// TwinCAT 3 PLC project CorteH2y3CX9265C4
// ProgramVersion: 3.1.4024.0
// libraries:
//   CmpBitmapPool, * (System)
//   Tc2_Standard, * (Beckhoff Automation GmbH)
//   Tc2_SUPS, * (Beckhoff Automation GmbH)
//   Tc2_System, * (Beckhoff Automation GmbH)
//   Tc2_Utilities, * (Beckhoff Automation GmbH)
//   Tc3_EventLogger, * (Beckhoff Automation GmbH)
//   Tc3_Module, * (Beckhoff Automation GmbH)
//   Visu Utils, * (System)
// project tree:
//   DUTs/ StrFuncParoEnviar.TcDUT (not stored), Str_Config_ADS_to_PLC.TcDUT (not stored), Str_HistTablasMySQL.TcDUT (not stored)
//   Events_Alarms/ Eventos_PLC.TcPOU (not stored), Events.TcPOU (not stored)
//   / GlobalTextList.TcGTLO, Lectura_PLC.TcTTO, PlcTask.TcTTO, VISU_TASK.TcTTO
//   GVLs/ Fecha_PLC.TcGVL (not stored), Lectura_PLCs.TcGVL (not stored), RegistroLocalDataBase.TcGVL, Var_Com_CH2_CH3.TcGVL
//   POUs/FBs/ fbLectura_a_PLC.TcPOU (not stored), fb_Funciones_Paro.TcPOU (not stored), FuncGeneralesCortHum3.TcPOU, FuncGeneralesCortHum2.TcPOU, TempParoAcumulad.TcPOU (not stored)
//   POUs/ Fecha_Hora_PLC.TcPOU (not stored), MAIN.TcPOU
//   POUs/Funciones comunes/ Utilidades.TcPOU
//   POUs/Lectura_a_PLC_Maestro/ Lectura_Maestro.TcPOU, MAIN_Orden_Lectura_PLCs.TcPOU (not stored)
//   POUs/PRGs_Nodos/ FuncParoNodoLocalCorteH3.TcPOU, FuncParoNodoRemote1CorteH2.TcPOU
//   VISUs/ Ajustes_CorteH2.TcVIS, Ajustes_CorteH3.TcVIS, DiagnosticoFB.TcVIS, HistTablaTablas_Ch2.TcVIS, HistTablaTablas_Ch3.TcVIS, Home_CortH2.TcVIS, Home_CortH3.TcVIS, Home_Sel_Maq.TcVIS, ImagePool.TcIPO (not stored), Modelo_Tabla_Ch2.TcVIS, Modelo_Tabla_Ch3.TcVIS, VisualizationManager.TcVMO (not stored), V_Emerg_Fin_Prod_Ch2.TcVIS, V_Emerg_Fin_Prod_Ch3.TcVIS
//   VISUs/IMAGENES/ Imagenes.TcIPO (not stored)
//   VISUs/Listas_Para_Desplegables/ FormatoTabla.TcTLO, EspesorTabla.TcTLO
// real-time tasks:
//   TASK PlcTask: cycle T#10ms, priority 20, ADS port 350
//   TASK VISU_TASK: cycle T#200000us, priority 30, ADS port 351
//   TASK Lectura_PLCs: cycle T#10ms, priority 1, ADS port 352
// I/O:
//   DEVICE Device 2 (EtherCAT), AmsNetId 5.146.101.196.3.1
//     Term 1 (EK1200) [EK1200-5000 EtherCAT Power supply (2A E-Bus)]
//       Term 2 (EL1859) [EL1859 8Ch. Dig. Input 24V, 3ms, 8Ch. Dig. Output 24V, 0.5A]
//       Term 3 (EK1110) [EK1110 EtherCAT extension]
//     Term 4 (EK1100) [EK1100 EtherCAT Coupler (2A E-Bus)]
//       Term 5 (EL1859) [EL1859 8Ch. Dig. Input 24V, 3ms, 8Ch. Dig. Output 24V, 0.5A]
//       Term 6 (EL9011) [EL9011 End Terminal]
// variable links:
//   CorteH2y3CX9265C4/CorteH2y3CX9265C4 Instance <-> Device 2 (EtherCAT)/Term 1 (EK1200)/Term 2 (EL1859)
//     PlcTask Inputs/MAIN.id0Local <-> Channel 1/Input
//     PlcTask Inputs/MAIN.id0Local @bit {1..7} <-> Channel {2..8}/Input  (7 links)
//     PlcTask Outputs/MAIN.od0Local @bit {1..7} <-> Channel {10..16}/Output  (7 links)
//     PlcTask Outputs/MAIN.od0Local <-> Channel 9/Output
//   CorteH2y3CX9265C4/CorteH2y3CX9265C4 Instance <-> Device 2 (EtherCAT)/Term 4 (EK1100)/Term 5 (EL1859)
//     PlcTask Inputs/MAIN.id0Remoto1 <-> Channel 1/Input
//     PlcTask Inputs/MAIN.id0Remoto1 @bit {1..7} <-> Channel {2..8}/Input  (7 links)
//     PlcTask Outputs/MAIN.od0Remoto1 @bit {1..7} <-> Channel {10..16}/Output  (7 links)
//     PlcTask Outputs/MAIN.od0Remoto1 <-> Channel 9/Output

CONFIGURATION CorteH2y3CX9265C4
    RESOURCE PLC ON TwinCAT3
        TASK Lectura_PLC(INTERVAL := T#10ms, PRIORITY := 1);
        TASK PlcTask(INTERVAL := T#10ms, PRIORITY := 20);
        TASK VISU_TASK(INTERVAL := T#200000us, PRIORITY := 30);
        PROGRAM MAIN_Orden_Lectura_PLCs WITH Lectura_PLC : MAIN_Orden_Lectura_PLCs;
        PROGRAM MAIN WITH PlcTask : MAIN;
        PROGRAM VisuElems_Visu_Prg WITH VISU_TASK : VisuElems.Visu_Prg;
    END_RESOURCE
END_CONFIGURATION

// ---- GVLs/RegistroLocalDataBase.TcGVL
{attribute 'qualified_only'}
VAR_GLOBAL
	aValoresTurnosAnt: ARRAY [0..50] OF StrFuncParoEnviar;//Cada fin de turno se envía los valores de la ultima tabla que ha psado y se queda guardado en esta array para enseñarlo por el Scada
END_VAR
VAR_GLOBAL PERSISTENT
	//Array para el histórico de las tablas enviado a la base de datos
	 aHistoricStrTablasCH2: ARRAY[0..100]OF Str_HistTablasMySQL;
	 aHistoricStrTablasCH3: ARRAY[0..100]OF Str_HistTablasMySQL;
END_VAR

// ---- GVLs/Var_Com_CH2_CH3.TcGVL
{attribute 'qualified_only'}
VAR_GLOBAL
	// Variables Escritura en PLC Maestro 
	aStringCom AT %MW2000: ARRAY[0..97] OF STRING;	//(1 string = 81 MW)
	aWordCom AT %MW10000: ARRAY[0..249] OF WORD;	//(1 Word = 1MW)
	aBoolCom AT %MB10250: ARRAY[0..499] OF BOOL;	//(1 Bool = 1MB)
	aTimeCom AT %MW10750: ARRAY[0..124] OF TIME;	//(1 Time = 4MW)
END_VAR

// ---- POUs/MAIN.TcPOU
PROGRAM MAIN
VAR
	// UPS variables persistentes
	fbUPS: FB_S_UPS_CX81xx;//Instancia de la UPS
	// Entradas
	id0Local   AT %I*: BYTE;
	id0Remoto1 AT %I*: BYTE;
	// Salidas
	od0Local   AT %Q*: BYTE;
	od0Remoto1 AT %Q*: BYTE;
	fbUtilidades: Utilidades;
END_VAR

fbUPS(iPLCPort:= 851,);
Fecha_Hora_PLC();
Events();
fbUtilidades();
FuncParoNodoLocalCorteH3();
FuncParoNodoRemote1CorteH2();

END_PROGRAM

// ---- POUs/Funciones comunes/Utilidades.TcPOU
FUNCTION_BLOCK Utilidades
VAR_INPUT
END_VAR
VAR_OUTPUT
END_VAR
VAR
sJustificaParoComun:STRING;
END_VAR

//Direccionamiento de variables para enviar 
Var_Com_CH2_CH3.aStringCom[62] := Fecha_PLC.StringDateHourMin;

END_FUNCTION_BLOCK

// ---- POUs/PRGs_Nodos/FuncParoNodoLocalCorteH3.TcPOU
PROGRAM FuncParoNodoLocalCorteH3
VAR
	Funci_CortHum3:fb_Funciones_Paro;
	FunGeneCortHum3: FuncGeneralesCortHum3;
	//Entradas Corte húmedo 4
	Ftc_CortHum3: BOOL;	
	ForzadoFtcCortHum3:BOOL;	
	Consenso_CortHum3: BOOL;
	//Entradas fotocelula 2 libre
	Ftc2_Libre: BOOL;
	ForzadoFtc2_Libre: BOOL;
	Consenso_Ftc2_Libre: BOOL;
	//Entradas fotocelula 3 libre
	Ftc3_Libre: BOOL;
	ForzadoFtc3_Libre: BOOL;
	Consenso_Ftc3_Libre: BOOL;
	//Entradas fotocelula 4 libre
	Ftc4_Libre: BOOL;
	ForzadoFtc4_Libre: BOOL;
	Consenso_Ftc4_Libre: BOOL;
	
//	Estructuras de las variables a enviar  
	CortHum3StrFuncParoEnviar:StrFuncParoEnviar;
	Ftc2StrFuncParoEnviar:StrFuncParoEnviar;	
	Ftc3StrFuncParoEnviar:StrFuncParoEnviar;
	Ftc4StrFuncParoEnviar:StrFuncParoEnviar;
	

END_VAR
VAR_INPUT
	sFormatoEleccionTabla:STRING;
	sModeloEleccionTabla:STRING;
	sEspesorEleccionTabla:STRING;
END_VAR
VAR RETAIN
END_VAR
VAR PERSISTENT 
	HMI_Tiempo_Offset_MParo:INT:=5;
	HMI_TiempoFiltradoFotocel:TIME:=T#2S;
// Modelo de la tabla y fecha cambio de modelo
	sModeloActualTabla:STRING;
	sFormatoActualTabla:STRING;
	sEspesorActualTabla:STRING;
	sFechaInicModeloTab:STRING;


END_VAR

//Funciones de paro para cada zona(Fotocelula)

//>>>>>>>>>>>>>>>>>>>>>>>>>>>>>>>>>>>>>>>>>>>>>         	Corte húmedo 4         <<<<<<<<<<<<<<<<<<<<<<<<<<<<<<<<<<<<<<<<<<<<<<<<<<<<<<<<<<
Funci_CortHum3(Fotocelula:=Ftc_CortHum3 OR ForzadoFtcCortHum3, 
					Tiempo_Offset_MParo:=HMI_Tiempo_Offset_MParo, 
					TiempoFiltradoFotocel:=HMI_TiempoFiltradoFotocel,
					_StrFuncParoEnviar => CortHum3StrFuncParoEnviar );
					
						
						
Direccionamiento_variables_com();
LinkadoEntradas();
FunGeneCortHum3(s_ModeloActualTabla => sModeloActualTabla,
				s_ModeloEleccionTabla => sModeloEleccionTabla,
				s_FechaInicModeloTab=>sFechaInicModeloTab,
				s_FormatoActualTabla=>sFormatoActualTabla,
				s_FormatoEleccionTabla=>sFormatoEleccionTabla,
				s_EspesorActualTabla=>sEspesorActualTabla,
				s_EspesorEleccionTabla=>sEspesorEleccionTabla);

ACTION Direccionamiento_variables_com:
// Direccionamiento de las variables a la marca que les corresponde donde después se leeran desde el plc maestro



//								>>>>>>>>>>>>>>>>>>>>>>>>>>>>      WORDS    <<<<<<<<<<<<<<<<<<<<<<<<<<<<<<<<

	Var_Com_CH2_CH3.aWordCom[0]:= INT_TO_WORD (CortHum3StrFuncParoEnviar.Cont_Piezas);	    //Contadores de cada fotocelula 
	Var_Com_CH2_CH3.aWordCom[1]:= INT_TO_WORD (Ftc2StrFuncParoEnviar.Cont_Piezas);		//Contadores de cada fotocelula 
	Var_Com_CH2_CH3.aWordCom[2]:= INT_TO_WORD (Ftc3StrFuncParoEnviar.Cont_Piezas);		//Contadores de cada fotocelula 
	Var_Com_CH2_CH3.aWordCom[3]:= INT_TO_WORD (Ftc4StrFuncParoEnviar.Cont_Piezas);		//Contadores de cada fotocelula 
	Var_Com_CH2_CH3.aWordCom[4]:= INT_TO_WORD (CortHum3StrFuncParoEnviar.Min_Parado_Ftc);			//Minutos actuales parado
	Var_Com_CH2_CH3.aWordCom[5]:= INT_TO_WORD (Ftc2StrFuncParoEnviar.Min_Parado_Ftc);			//Minutos actuales parado
	Var_Com_CH2_CH3.aWordCom[6]:= INT_TO_WORD (Ftc3StrFuncParoEnviar.Min_Parado_Ftc);			//Minutos actuales parado
	Var_Com_CH2_CH3.aWordCom[7]:= INT_TO_WORD (Ftc4StrFuncParoEnviar.Min_Parado_Ftc);			//Minutos actuales parado
	
	
	
//                           	>>>>>>>>>>>>>>>>>>>>>>>>>>>>      TIME   <<<<<<<<<<<<<<<<<<<<<<<<<<<<<<<<
	
	
	Var_Com_CH2_CH3.aTimeCom[0]:=  CortHum3StrFuncParoEnviar.t_Entre_Piez_Ftc; 			//Tiempo entre piezas
	Var_Com_CH2_CH3.aTimeCom[1]:=  Ftc2StrFuncParoEnviar.t_Entre_Piez_Ftc;			//Tiempo entre piezas
	Var_Com_CH2_CH3.aTimeCom[2]:= Ftc3StrFuncParoEnviar.t_Entre_Piez_Ftc;				//Tiempo entre piezas
	Var_Com_CH2_CH3.aTimeCom[3]:= Ftc4StrFuncParoEnviar.t_Entre_Piez_Ftc;				//Tiempo entre piezas
	Var_Com_CH2_CH3.aTimeCom[4]:= CortHum3StrFuncParoEnviar.t_Entr_Piez_Ante_Ftc; 		//Tiempo entre piezas anterior
	Var_Com_CH2_CH3.aTimeCom[5]:= Ftc2StrFuncParoEnviar.t_Entr_Piez_Ante_Ftc; 		//Tiempo entre piezas anterior
	Var_Com_CH2_CH3.aTimeCom[6]:= Ftc3StrFuncParoEnviar.t_Entr_Piez_Ante_Ftc; 		//Tiempo entre piezas anterior
	Var_Com_CH2_CH3.aTimeCom[7]:= Ftc4StrFuncParoEnviar.t_Entr_Piez_Ante_Ftc; 		//Tiempo entre piezas anterior
	
	
	
	
//                           	>>>>>>>>>>>>>>>>>>>>>>>>>>>>      STRING  <<<<<<<<<<<<<<<<<<<<<<<<<<<<<<<<
    Var_Com_CH2_CH3.aStringCom[0] := CortHum3StrFuncParoEnviar.H_InParo_Ftc;         //Hora inicio paro 
	Var_Com_CH2_CH3.aStringCom[1] := Ftc2StrFuncParoEnviar.H_InParo_Ftc;         //Hora inicio paro 
	Var_Com_CH2_CH3.aStringCom[2] := Ftc3StrFuncParoEnviar.H_InParo_Ftc;         //Hora inicio paro 
	Var_Com_CH2_CH3.aStringCom[3] := Ftc4StrFuncParoEnviar.H_InParo_Ftc;         //Hora inicio paro 
	Var_Com_CH2_CH3.aStringCom[4] := CortHum3StrFuncParoEnviar.H_FinParo_Ftc;        //Hora Fin paro 
	Var_Com_CH2_CH3.aStringCom[5] := Ftc2StrFuncParoEnviar.H_FinParo_Ftc;        //Hora Fin paro 
	Var_Com_CH2_CH3.aStringCom[6] := Ftc3StrFuncParoEnviar.H_FinParo_Ftc;        //Hora Fin paro 
	Var_Com_CH2_CH3.aStringCom[7] := Ftc4StrFuncParoEnviar.H_FinParo_Ftc;        //Hora Fin paro 
	Var_Com_CH2_CH3.aStringCom[8] := CortHum3StrFuncParoEnviar.S_Justi_Paro_Ftc;		//Justificación del paro
	Var_Com_CH2_CH3.aStringCom[9] := Ftc2StrFuncParoEnviar.S_Justi_Paro_Ftc;		//Justificación del paro
	Var_Com_CH2_CH3.aStringCom[10] := Ftc3StrFuncParoEnviar.S_Justi_Paro_Ftc;		//Justificación del paro
	Var_Com_CH2_CH3.aStringCom[11] := Ftc4StrFuncParoEnviar.S_Justi_Paro_Ftc;		//Justificación del paro
	
	
//                           	>>>>>>>>>>>>>>>>>>>>>>>>>>>>      Bool  <<<<<<<<<<<<<<<<<<<<<<<<<<<<<<<<	

	Var_Com_CH2_CH3.aBoolCom[0] := CortHum3StrFuncParoEnviar.Fotocelula;						//Fotocelula Real
	Var_Com_CH2_CH3.aBoolCom[1] := Ftc2StrFuncParoEnviar.Fotocelula;						//Fotocelula Real
	Var_Com_CH2_CH3.aBoolCom[2] := Ftc3StrFuncParoEnviar.Fotocelula;						//Fotocelula Real
	Var_Com_CH2_CH3.aBoolCom[3] := Ftc4StrFuncParoEnviar.Fotocelula;						//Fotocelula Real
	Var_Com_CH2_CH3.aBoolCom[4] := CortHum3StrFuncParoEnviar.MParo_Ftc;				//Marca de paro 
	Var_Com_CH2_CH3.aBoolCom[5] := Ftc2StrFuncParoEnviar.MParo_Ftc;				//Marca de paro 
	Var_Com_CH2_CH3.aBoolCom[6] := Ftc3StrFuncParoEnviar.MParo_Ftc;				//Marca de paro 
	Var_Com_CH2_CH3.aBoolCom[7] := Ftc4StrFuncParoEnviar.MParo_Ftc;				//Marca de paro 
	Var_Com_CH2_CH3.aBoolCom[8] := CortHum3StrFuncParoEnviar.M_SinParo_Ftc;			//Marca de sin paro activo
	Var_Com_CH2_CH3.aBoolCom[9] := Ftc2StrFuncParoEnviar.M_SinParo_Ftc;			//Marca de sin paro activo
	Var_Com_CH2_CH3.aBoolCom[10] := Ftc3StrFuncParoEnviar.M_SinParo_Ftc;			//Marca de sin paro activo
	Var_Com_CH2_CH3.aBoolCom[11] := Ftc4StrFuncParoEnviar.M_SinParo_Ftc;			//Marca de sin paro activo
	Var_Com_CH2_CH3.aBoolCom[12] := CortHum3StrFuncParoEnviar.tFiltro_up_Ftc;			//Q Temp Up Filtro Fotocelulas
	Var_Com_CH2_CH3.aBoolCom[13] := Ftc2StrFuncParoEnviar.tFiltro_up_Ftc;			//Q Temp Up Filtro Fotocelulas
	Var_Com_CH2_CH3.aBoolCom[14] := Ftc3StrFuncParoEnviar.tFiltro_up_Ftc;			//Q Temp Up Filtro Fotocelulas
	Var_Com_CH2_CH3.aBoolCom[15] := Ftc4StrFuncParoEnviar.tFiltro_up_Ftc;			//Q Temp Up Filtro Fotocelulas
	Var_Com_CH2_CH3.aBoolCom[16] := CortHum3StrFuncParoEnviar.tFiltro_down_Ftc;		//Q Temp Down Filtro Fotocelulas
	Var_Com_CH2_CH3.aBoolCom[17] := Ftc2StrFuncParoEnviar.tFiltro_down_Ftc;		//Q Temp Down Filtro Fotocelulas
	Var_Com_CH2_CH3.aBoolCom[18] := Ftc3StrFuncParoEnviar.tFiltro_down_Ftc;		//Q Temp Down Filtro Fotocelulas
	Var_Com_CH2_CH3.aBoolCom[19] := Ftc4StrFuncParoEnviar.tFiltro_down_Ftc;		//Q Temp Down Filtro Fotocelulas
END_ACTION

ACTION LinkadoEntradas:
// Linkado entradas

Ftc_CortHum3:=      main.id0Local.0;
Consenso_CortHum3:= TRUE;//main.id0Remoto1.1;


Ftc2_Libre:=      main.id0Local.2;
Consenso_Ftc3_Libre:= TRUE;// main.id0Remoto1.3;


Ftc3_Libre:=      main.id0Local.4;
Consenso_Ftc3_Libre:= TRUE;// main.id0Remoto1.5;


Ftc4_Libre:=      main.id0Local.6;
Consenso_Ftc4_Libre:= TRUE;// main.id0Remoto1.7;
END_ACTION

PROPERTY PUBLIC s_JustifParoCH3 : STRING
GET
s_JustifParoCH3:= Funci_CortHum3.S_Justi_Paro_Ftc;
END_GET
SET
Funci_CortHum3.S_Justi_Paro_Ftc:=s_JustifParoCH3;
END_SET
END_PROPERTY

END_PROGRAM

// ---- POUs/FBs/FuncGeneralesCortHum3.TcPOU
FUNCTION_BLOCK FuncGeneralesCortHum3
VAR_INPUT
IndexListFormatoTabla:INT;
IndexJustificacionParo:INT;
IndexListEspesorTabla:INT;
END_VAR
VAR_OUTPUT
	//Modelo dividido en strings para DataBase
	s_ModeloActualTabla:STRING;
	s_FormatoActualTabla:STRING;
	s_EspesorActualTabla:STRING;
	s_ModeloEleccionTabla:STRING;
	s_FormatoEleccionTabla:STRING;
	s_EspesorEleccionTabla:STRING;
	//Comunes
	s_JustificaParoComun:STRING;
	s_FechaInicModeloTab:STRING;
END_VAR
VAR
	Reset_Fin_Prod:BOOL;
	P_FinProduccion:BOOL;
	P_EscribirModelo:BOOL;
	pul_Justif_Paro:BOOL;
	EscribeHistoricTablas:BOOL;
	FlancFiltUpFtcEscHistTab:R_TRIG;
	Cont1:INT;
	Cont2:INT;
	Cont3:INT;
	Cont4:INT;
END_VAR
VAR PERSISTENT 
	PointerHistTablas:INT;
END_VAR

//                             >>>>>>>>>>>>>>>> Modelo de la tabla <<<<<<<<<<<<<<<<<

//Fin de producción 		
IF P_FinProduccion THEN 
Fin_Produccion();
END_IF;
IF P_EscribirModelo THEN
	ListFormatoTabla(); 
	ListadoEspesorTabla();
	Inicio_Nuevo_Modelo();
	
END_IF


//Envío de la linea de la tabla para el historico de control producción en el HMI del operario
 IF FlancFiltUpFtcEscHistTab.Q THEN 
	 EscStrHistoricoTablas();
 END_IF


Direccionamiento_variables_com();
FlancFiltUpFtcEscHistTab(CLK := FuncParoNodoLocalCorteH3.Funci_CortHum3.tFiltro_up_Ftc.Q);

ACTION Direccionamiento_variables_com:
	//                           	>>>>>>>>>>>>>>>>>>>>>>>>>>>>      STRING      <<<<<<<<<<<<<<<<<<<<<<<<<<<<<<<<
    Var_Com_CH2_CH3.aStringCom[80] := s_ModeloActualTabla;
	Var_Com_CH2_CH3.aStringCom[81] := s_FormatoActualTabla;
	Var_Com_CH2_CH3.aStringCom[82] := s_EspesorActualTabla;
	Var_Com_CH2_CH3.aStringCom[83] := s_FechaInicModeloTab;
END_ACTION

METHOD EscStrHistoricoTablas : BOOL
VAR_INPUT
END_VAR
// Recorre todas las lineas de la tabla una posición y añade la nueva tabla en la linea 0 para mayor coodidad al visulizar

FOR PointerHistTablas := 100 TO 1 BY -1 DO 
	RegistroLocalDataBase.aHistoricStrTablasCH3[PointerHistTablas].ID := RegistroLocalDataBase.aHistoricStrTablasCH3[PointerHistTablas-1].ID;
	RegistroLocalDataBase.aHistoricStrTablasCH3[PointerHistTablas].Fecha := RegistroLocalDataBase.aHistoricStrTablasCH3[PointerHistTablas-1].Fecha;
	RegistroLocalDataBase.aHistoricStrTablasCH3[PointerHistTablas].Modelo := RegistroLocalDataBase.aHistoricStrTablasCH3[PointerHistTablas-1].Modelo;
	RegistroLocalDataBase.aHistoricStrTablasCH3[PointerHistTablas].Formato := RegistroLocalDataBase.aHistoricStrTablasCH3[PointerHistTablas-1].Formato;
	RegistroLocalDataBase.aHistoricStrTablasCH3[PointerHistTablas].Espesor :=RegistroLocalDataBase.aHistoricStrTablasCH3[PointerHistTablas-1].Espesor;
	RegistroLocalDataBase.aHistoricStrTablasCH3[PointerHistTablas].Maquina := RegistroLocalDataBase.aHistoricStrTablasCH3[PointerHistTablas-1].Maquina;
	RegistroLocalDataBase.aHistoricStrTablasCH3[PointerHistTablas].Cont_Piezas := RegistroLocalDataBase.aHistoricStrTablasCH3[PointerHistTablas-1].Cont_Piezas;
	RegistroLocalDataBase.aHistoricStrTablasCH3[PointerHistTablas].t_Entre_Piez_Ftc := RegistroLocalDataBase.aHistoricStrTablasCH3[PointerHistTablas-1].t_Entre_Piez_Ftc;
	RegistroLocalDataBase.aHistoricStrTablasCH3[PointerHistTablas].S_Justi_Paro_Ftc := RegistroLocalDataBase.aHistoricStrTablasCH3[PointerHistTablas-1].S_Justi_Paro_Ftc;
	
END_FOR
//Estructura de la array de la tabla para visualizar el historico de la tablas pasadas
RegistroLocalDataBase.aHistoricStrTablasCH3[0].ID := PointerHistTablas;
RegistroLocalDataBase.aHistoricStrTablasCH3[0].Fecha := Fecha_PLC.StringDateHourMin;
RegistroLocalDataBase.aHistoricStrTablasCH3[0].Modelo := FuncParoNodoLocalCorteH3.sModeloActualTabla;
RegistroLocalDataBase.aHistoricStrTablasCH3[0].Formato := FuncParoNodoLocalCorteH3.sFormatoActualTabla;
RegistroLocalDataBase.aHistoricStrTablasCH3[0].Espesor :=FuncParoNodoLocalCorteH3.sEspesorActualTabla;
RegistroLocalDataBase.aHistoricStrTablasCH3[0].Maquina := 'Corte húmedo 2';
RegistroLocalDataBase.aHistoricStrTablasCH3[0].Cont_Piezas := FuncParoNodoLocalCorteH3.Funci_CortHum3.Cont_Piezas_Ftc;
RegistroLocalDataBase.aHistoricStrTablasCH3[0].t_Entre_Piez_Ftc := FuncParoNodoLocalCorteH3.Funci_CortHum3.t_Entre_Piez_Ftc;
RegistroLocalDataBase.aHistoricStrTablasCH3[0].S_Justi_Paro_Ftc := FuncParoNodoLocalCorteH3.Funci_CortHum3.S_Justi_Paro_Ftc;
END_METHOD

METHOD Fin_Produccion : BOOL
VAR_INPUT	
END_VAR
var
	Puls_Fin_Produccion:BOOL;	
END_VAR
//Valores por defecto del modelo y fecha de inicio modelo

s_ModeloActualTabla:= 'Sin modelo de pieza';
s_ModeloEleccionTabla:= 'Sin modelo de pieza';
s_FormatoActualTabla:= 'Sin modelo de pieza';
s_FormatoEleccionTabla:= 'Sin modelo de pieza';
s_EspesorActualTabla:= 'Sin modelo de pieza';
s_EspesorEleccionTabla:= 'Sin modelo de pieza';
s_FechaInicModeloTab:= 'Sin modelo de pieza';
 
//Reset contador de piezas 
FuncParoNodoLocalCorteH3.Funci_CortHum3.Fin_Produccion();
END_METHOD

METHOD Inicio_Nuevo_Modelo : BOOL
VAR_INPUT
END_VAR
VAR
END_VAR

// Envías la fecha de inicio modelo de tabla 
s_FechaInicModeloTab:=Fecha_PLC.Mes_Dia_Hora_Min_Real;

//Envías el modelo de la tabla de la variable preelección  
s_ModeloActualTabla:=s_ModeloEleccionTabla;
s_FormatoActualTabla:=s_FormatoEleccionTabla;
s_EspesorActualTabla:= s_EspesorEleccionTabla;
END_METHOD

METHOD ListadoEspesorTabla : BOOL
VAR_INPUT
END_VAR
// Función para poder realizar el desplegable de espesor de la tabla en el Visu
IF IndexListEspesorTabla <> 5 THEN 
	IF IndexListEspesorTabla = 1 THEN 
		s_EspesorEleccionTabla:='3';
	END_IF
	IF IndexListEspesorTabla = 2 THEN 
		s_EspesorEleccionTabla:='6';
	END_IF
	IF IndexListEspesorTabla = 3 THEN 
		s_EspesorEleccionTabla:='12';
	END_IF
	IF IndexListEspesorTabla = 4 THEN 
		s_EspesorEleccionTabla:='20';
	END_IF
END_IF
END_METHOD

METHOD ListadoJustificacionParo : BOOL
VAR_INPUT
END_VAR
// Envío Justificación de los paros prefijados

(*Listado:  0:Sin asignar
			1: Descanso
			2: Avería
			3: Cambio de discos 
			4: Cambio de formato
			5: Cambio caballete/bandeja 
			6: Mantenimiento
			7: Falta material 
			8: Preparación material 
			9: Limpieza fin de turno 
			10: Ninguno de la lista			 
*)
//Descanso
IF IndexJustificacionParo = 1 THEN 
	FuncParoNodoLocalCorteH3.s_JustifParoCH3 := 'Descanso';
END_IF
// Avería 
IF IndexJustificacionParo = 2 THEN 
	FuncParoNodoLocalCorteH3.s_JustifParoCH3 := 'Avería';
END_IF
//Cambio de discos 
IF IndexJustificacionParo = 3 THEN 
	FuncParoNodoLocalCorteH3.s_JustifParoCH3 := 'Cambio de discos';
END_IF
// Cambio de formato
IF IndexJustificacionParo = 4 THEN 
	FuncParoNodoLocalCorteH3.s_JustifParoCH3 := 'Cambio de formato';
END_IF
//Cambio caballete/bandeja
IF IndexJustificacionParo = 5 THEN 
	FuncParoNodoLocalCorteH3.s_JustifParoCH3 := 'Cambio caballete/bandeja';
END_IF
// Mantenimiento
IF IndexJustificacionParo = 6 THEN 
	FuncParoNodoLocalCorteH3.s_JustifParoCH3 := 'Mantenimiento';
END_IF
// Falta de material 
IF IndexJustificacionParo = 7 THEN 
	FuncParoNodoLocalCorteH3.s_JustifParoCH3 := 'Falta de material';
END_IF
//Preparación de material 
IF IndexJustificacionParo = 8 THEN 
	FuncParoNodoLocalCorteH3.s_JustifParoCH3 := 'Preparación de material';
END_IF
// Limpieza fin de turno
IF IndexJustificacionParo = 9 THEN 
	FuncParoNodoLocalCorteH3.s_JustifParoCH3 := 'Limpieza fin de turno';
END_IF
// No está en la lista
IF IndexJustificacionParo = 10 THEN 
	FuncParoNodoLocalCorteH3.s_JustifParoCH3 := 'ESCRIBE AQUÍ LA JUSTIFICACIÓN DEL PARO';
END_IF
END_METHOD

METHOD ListFormatoTabla : BOOL
VAR_INPUT
END_VAR
// Función para poder realizar el desplegable de formato de la tabla en el Visu
IF IndexListFormatoTabla <> 8 THEN 
	IF IndexListFormatoTabla = 1 THEN 
		s_FormatoEleccionTabla:='3200 X 1500';
		Cont1:=Cont1+1;
	END_IF
	IF IndexListFormatoTabla = 2 THEN 
		s_FormatoEleccionTabla:='3600 X 1200';
		Cont2:=Cont2+1;
	END_IF
	IF IndexListFormatoTabla = 3 THEN 
		s_FormatoEleccionTabla:='1800 X 1200';
	END_IF
	IF IndexListFormatoTabla = 4 THEN 
		s_FormatoEleccionTabla:='3000 X 1000';
	END_IF
	IF IndexListFormatoTabla = 5 THEN 
		s_FormatoEleccionTabla:='2600 X 1500';
	END_IF
	IF IndexListFormatoTabla = 6 THEN 
		s_FormatoEleccionTabla:='800 X 700';
	END_IF
	IF IndexListFormatoTabla = 7 THEN 
		s_FormatoEleccionTabla:='2700 X 1000';
	END_IF
END_IF
END_METHOD

END_FUNCTION_BLOCK

// ---- POUs/PRGs_Nodos/FuncParoNodoRemote1CorteH2.TcPOU
PROGRAM FuncParoNodoRemote1CorteH2
VAR
	Funci_CortHum2:fb_Funciones_Paro;
	FunGeneCortHum2: FuncGeneralesCortHum2;
	//Entradas Corte húmedo 4
	Ftc_CortHum2: BOOL;	
	ForzadoFtcCortHum2:BOOL;	
	Consenso_CortHum2: BOOL;
	//Entradas fotocelula 2 libre
	Ftc2_Libre: BOOL;
	ForzadoFtc2_Libre: BOOL;
	Consenso_Ftc2_Libre: BOOL;
	//Entradas fotocelula 3 libre
	Ftc3_Libre: BOOL;
	ForzadoFtc3_Libre: BOOL;
	Consenso_Ftc3_Libre: BOOL;
	//Entradas fotocelula 4 libre
	Ftc4_Libre: BOOL;
	ForzadoFtc4_Libre: BOOL;
	Consenso_Ftc4_Libre: BOOL;
	
//	Estructuras de las variables a enviar  
	CortHum2StrFuncParoEnviar:StrFuncParoEnviar;
	Ftc2StrFuncParoEnviar:StrFuncParoEnviar;	
	Ftc3StrFuncParoEnviar:StrFuncParoEnviar;
	Ftc4StrFuncParoEnviar:StrFuncParoEnviar;
	

END_VAR
VAR_INPUT
	sFormatoEleccionTabla:STRING;
	sModeloEleccionTabla:STRING;
	sEspesorEleccionTabla:STRING;
END_VAR
VAR RETAIN
END_VAR
VAR PERSISTENT 
	HMI_Tiempo_Offset_MParo:INT:=5;
	HMI_TiempoFiltradoFotocel:TIME:=T#2S;
// Modelo de la tabla y fecha cambio de modelo
	sModeloActualTabla:STRING;
	sFormatoActualTabla:STRING;
	sEspesorActualTabla:STRING;
	sFechaInicModeloTab:STRING;


END_VAR

//Funciones de paro para cada zona(Fotocelula)

//>>>>>>>>>>>>>>>>>>>>>>>>>>>>>>>>>>>>>>>>>>>>>         	Corte húmedo 4         <<<<<<<<<<<<<<<<<<<<<<<<<<<<<<<<<<<<<<<<<<<<<<<<<<<<<<<<<<
Funci_CortHum2(Fotocelula:=Ftc_CortHum2 OR ForzadoFtcCortHum2, 
					Tiempo_Offset_MParo:=HMI_Tiempo_Offset_MParo, 
					TiempoFiltradoFotocel:=HMI_TiempoFiltradoFotocel,
					_StrFuncParoEnviar => CortHum2StrFuncParoEnviar );
					
						
						
Direccionamiento_variables_com();
LinkadoEntradas();
FunGeneCortHum2(s_ModeloActualTabla => sModeloActualTabla,s_ModeloEleccionTabla => sModeloEleccionTabla,s_FechaInicModeloTab=>sFechaInicModeloTab,s_FormatoActualTabla=>sFormatoActualTabla,s_FormatoEleccionTabla=>sFormatoEleccionTabla,s_EspesorActualTabla=>sEspesorActualTabla,s_EspesorEleccionTabla=>sEspesorEleccionTabla);

ACTION Direccionamiento_variables_com:
// Direccionamiento de las variables a la marca que les corresponde donde despés se leeran desde el plc maestro



//								>>>>>>>>>>>>>>>>>>>>>>>>>>>>      WORDS    <<<<<<<<<<<<<<<<<<<<<<<<<<<<<<<<

	Var_Com_CH2_CH3.aWordCom[50]:= INT_TO_WORD (CortHum2StrFuncParoEnviar.Cont_Piezas);	    //Contadores de cada fotocelula 
	Var_Com_CH2_CH3.aWordCom[51]:= INT_TO_WORD (Ftc2StrFuncParoEnviar.Cont_Piezas);		//Contadores de cada fotocelula 
	Var_Com_CH2_CH3.aWordCom[52]:= INT_TO_WORD (Ftc3StrFuncParoEnviar.Cont_Piezas);		//Contadores de cada fotocelula 
	Var_Com_CH2_CH3.aWordCom[53]:= INT_TO_WORD (Ftc4StrFuncParoEnviar.Cont_Piezas);		//Contadores de cada fotocelula 
	Var_Com_CH2_CH3.aWordCom[54]:= INT_TO_WORD (CortHum2StrFuncParoEnviar.Min_Parado_Ftc);			//Minutos actuales parado
	Var_Com_CH2_CH3.aWordCom[55]:= INT_TO_WORD (Ftc2StrFuncParoEnviar.Min_Parado_Ftc);			//Minutos actuales parado
	Var_Com_CH2_CH3.aWordCom[56]:= INT_TO_WORD (Ftc3StrFuncParoEnviar.Min_Parado_Ftc);			//Minutos actuales parado
	Var_Com_CH2_CH3.aWordCom[57]:= INT_TO_WORD (Ftc4StrFuncParoEnviar.Min_Parado_Ftc);			//Minutos actuales parado
	
	
	
//                           	>>>>>>>>>>>>>>>>>>>>>>>>>>>>      TIME   <<<<<<<<<<<<<<<<<<<<<<<<<<<<<<<<
	
	
	Var_Com_CH2_CH3.aTimeCom[25]:=  CortHum2StrFuncParoEnviar.t_Entre_Piez_Ftc; 			//Tiempo entre piezas
	Var_Com_CH2_CH3.aTimeCom[26]:=  Ftc2StrFuncParoEnviar.t_Entre_Piez_Ftc;			//Tiempo entre piezas
	Var_Com_CH2_CH3.aTimeCom[27]:= Ftc3StrFuncParoEnviar.t_Entre_Piez_Ftc;				//Tiempo entre piezas
	Var_Com_CH2_CH3.aTimeCom[28]:= Ftc4StrFuncParoEnviar.t_Entre_Piez_Ftc;				//Tiempo entre piezas
	Var_Com_CH2_CH3.aTimeCom[29]:= CortHum2StrFuncParoEnviar.t_Entr_Piez_Ante_Ftc; 		//Tiempo entre piezas anterior
	Var_Com_CH2_CH3.aTimeCom[30]:= Ftc2StrFuncParoEnviar.t_Entr_Piez_Ante_Ftc; 		//Tiempo entre piezas anterior
	Var_Com_CH2_CH3.aTimeCom[31]:= Ftc3StrFuncParoEnviar.t_Entr_Piez_Ante_Ftc; 		//Tiempo entre piezas anterior
	Var_Com_CH2_CH3.aTimeCom[32]:= Ftc4StrFuncParoEnviar.t_Entr_Piez_Ante_Ftc; 		//Tiempo entre piezas anterior
	
	
	
	
//                           	>>>>>>>>>>>>>>>>>>>>>>>>>>>>      STRING  <<<<<<<<<<<<<<<<<<<<<<<<<<<<<<<<
    Var_Com_CH2_CH3.aStringCom[20] := CortHum2StrFuncParoEnviar.H_InParo_Ftc;         //Hora inicio paro 
	Var_Com_CH2_CH3.aStringCom[21] := Ftc2StrFuncParoEnviar.H_InParo_Ftc;         //Hora inicio paro 
	Var_Com_CH2_CH3.aStringCom[22] := Ftc3StrFuncParoEnviar.H_InParo_Ftc;         //Hora inicio paro 
	Var_Com_CH2_CH3.aStringCom[23] := Ftc4StrFuncParoEnviar.H_InParo_Ftc;         //Hora inicio paro 
	Var_Com_CH2_CH3.aStringCom[24] := CortHum2StrFuncParoEnviar.H_FinParo_Ftc;        //Hora Fin paro 
	Var_Com_CH2_CH3.aStringCom[25] := Ftc2StrFuncParoEnviar.H_FinParo_Ftc;        //Hora Fin paro 
	Var_Com_CH2_CH3.aStringCom[26] := Ftc3StrFuncParoEnviar.H_FinParo_Ftc;        //Hora Fin paro 
	Var_Com_CH2_CH3.aStringCom[27] := Ftc4StrFuncParoEnviar.H_FinParo_Ftc;        //Hora Fin paro 
	Var_Com_CH2_CH3.aStringCom[28] := CortHum2StrFuncParoEnviar.S_Justi_Paro_Ftc;		//Justificación del paro
	Var_Com_CH2_CH3.aStringCom[29] := Ftc2StrFuncParoEnviar.S_Justi_Paro_Ftc;		//Justificación del paro
	Var_Com_CH2_CH3.aStringCom[30] := Ftc3StrFuncParoEnviar.S_Justi_Paro_Ftc;		//Justificación del paro
	Var_Com_CH2_CH3.aStringCom[31] := Ftc4StrFuncParoEnviar.S_Justi_Paro_Ftc;		//Justificación del paro
	
	
//                           	>>>>>>>>>>>>>>>>>>>>>>>>>>>>      Bool  <<<<<<<<<<<<<<<<<<<<<<<<<<<<<<<<	

	Var_Com_CH2_CH3.aBoolCom[99] := CortHum2StrFuncParoEnviar.Fotocelula;						//Fotocelula Real
	Var_Com_CH2_CH3.aBoolCom[100] := Ftc2StrFuncParoEnviar.Fotocelula;						//Fotocelula Real
	Var_Com_CH2_CH3.aBoolCom[101] := Ftc3StrFuncParoEnviar.Fotocelula;						//Fotocelula Real
	Var_Com_CH2_CH3.aBoolCom[102] := Ftc4StrFuncParoEnviar.Fotocelula;						//Fotocelula Real
	Var_Com_CH2_CH3.aBoolCom[103] := CortHum2StrFuncParoEnviar.MParo_Ftc;				//Marca de paro 
	Var_Com_CH2_CH3.aBoolCom[104] := Ftc2StrFuncParoEnviar.MParo_Ftc;				//Marca de paro 
	Var_Com_CH2_CH3.aBoolCom[105] := Ftc3StrFuncParoEnviar.MParo_Ftc;				//Marca de paro 
	Var_Com_CH2_CH3.aBoolCom[106] := Ftc4StrFuncParoEnviar.MParo_Ftc;				//Marca de paro 
	Var_Com_CH2_CH3.aBoolCom[107] := CortHum2StrFuncParoEnviar.M_SinParo_Ftc;			//Marca de sin paro activo
	Var_Com_CH2_CH3.aBoolCom[108] := Ftc2StrFuncParoEnviar.M_SinParo_Ftc;			//Marca de sin paro activo
	Var_Com_CH2_CH3.aBoolCom[109] := Ftc3StrFuncParoEnviar.M_SinParo_Ftc;			//Marca de sin paro activo
	Var_Com_CH2_CH3.aBoolCom[110] := Ftc4StrFuncParoEnviar.M_SinParo_Ftc;			//Marca de sin paro activo
	Var_Com_CH2_CH3.aBoolCom[111] := CortHum2StrFuncParoEnviar.tFiltro_up_Ftc;			//Q Temp Up Filtro Fotocelulas
	Var_Com_CH2_CH3.aBoolCom[112] := Ftc2StrFuncParoEnviar.tFiltro_up_Ftc;			//Q Temp Up Filtro Fotocelulas
	Var_Com_CH2_CH3.aBoolCom[113] := Ftc3StrFuncParoEnviar.tFiltro_up_Ftc;			//Q Temp Up Filtro Fotocelulas
	Var_Com_CH2_CH3.aBoolCom[114] := Ftc4StrFuncParoEnviar.tFiltro_up_Ftc;			//Q Temp Up Filtro Fotocelulas
	Var_Com_CH2_CH3.aBoolCom[115] := CortHum2StrFuncParoEnviar.tFiltro_down_Ftc;		//Q Temp Down Filtro Fotocelulas
	Var_Com_CH2_CH3.aBoolCom[116] := Ftc2StrFuncParoEnviar.tFiltro_down_Ftc;		//Q Temp Down Filtro Fotocelulas
	Var_Com_CH2_CH3.aBoolCom[117] := Ftc3StrFuncParoEnviar.tFiltro_down_Ftc;		//Q Temp Down Filtro Fotocelulas
	Var_Com_CH2_CH3.aBoolCom[118] := Ftc4StrFuncParoEnviar.tFiltro_down_Ftc;		//Q Temp Down Filtro Fotocelulas
END_ACTION

ACTION LinkadoEntradas:





// Linkado entradas

Ftc_CortHum2:=      main.id0Remoto1.0;
Consenso_CortHum2:= TRUE;//main.id0Remoto1.1;


Ftc2_Libre:=      main.id0Remoto1.2;
Consenso_Ftc3_Libre:= TRUE;// main.id0Remoto1.3;


Ftc3_Libre:=      main.id0Remoto1.4;
Consenso_Ftc3_Libre:= TRUE;// main.id0Remoto1.5;


Ftc4_Libre:=      main.id0Remoto1.6;
Consenso_Ftc4_Libre:= TRUE;// main.id0Remoto1.7;
END_ACTION

PROPERTY PUBLIC s_JustifParoCH2 : STRING
GET
s_JustifParoCH2:= Funci_CortHum2.S_Justi_Paro_Ftc;
END_GET
SET
Funci_CortHum2.S_Justi_Paro_Ftc:=s_JustifParoCH2;
END_SET
END_PROPERTY

END_PROGRAM

// ---- POUs/FBs/FuncGeneralesCortHum2.TcPOU
FUNCTION_BLOCK FuncGeneralesCortHum2
VAR_INPUT
IndexListFormatoTabla:INT;
IndexJustificacionParo:INT;
IndexListEspesorTabla:INT;
END_VAR
VAR_OUTPUT
	//Modelo dividido en strings para DataBase
	s_ModeloActualTabla:STRING;
	s_FormatoActualTabla:STRING;
	s_EspesorActualTabla:STRING;
	s_ModeloEleccionTabla:STRING;
	s_FormatoEleccionTabla:STRING;
	s_EspesorEleccionTabla:STRING;
	//Comunes
	s_JustificaParoComun:STRING;
	s_FechaInicModeloTab:STRING;
END_VAR
VAR
	Reset_Fin_Prod:BOOL;
	P_FinProduccion:BOOL;
	P_EscribirModelo:BOOL;
	pul_Justif_Paro:BOOL;
	EscribeHistoricTablas:BOOL;
	FlancFiltUpFtcEscHistTab:R_TRIG;
	Cont1:INT;
	Cont2:INT;
	Cont3:INT;
	Cont4:INT;
END_VAR
VAR PERSISTENT 
	PointerHistTablas:INT;
END_VAR

//                             >>>>>>>>>>>>>>>> Modelo de la tabla <<<<<<<<<<<<<<<<<

//Fin de producción 		
IF P_FinProduccion THEN 
Fin_Produccion();
END_IF;
IF P_EscribirModelo THEN
	ListFormatoTabla(); 
	ListadoEspesorTabla();
	Inicio_Nuevo_Modelo();
	
END_IF


//Envío de la linea de la tabla para el historico de control producción en el HMI del operario
 IF FlancFiltUpFtcEscHistTab.Q THEN 
	 EscStrHistoricoTablas();
 END_IF


Direccionamiento_variables_com();
FlancFiltUpFtcEscHistTab(CLK := FuncParoNodoRemote1CorteH2.Funci_CortHum2.tFiltro_up_Ftc.Q);

ACTION Direccionamiento_variables_com:
	//                           	>>>>>>>>>>>>>>>>>>>>>>>>>>>>      STRING      <<<<<<<<<<<<<<<<<<<<<<<<<<<<<<<<
    Var_Com_CH2_CH3.aStringCom[84] := s_ModeloActualTabla;
	Var_Com_CH2_CH3.aStringCom[85] := s_FormatoActualTabla;
	Var_Com_CH2_CH3.aStringCom[86] := s_EspesorActualTabla;
	Var_Com_CH2_CH3.aStringCom[87] := s_FechaInicModeloTab;
END_ACTION

METHOD EscStrHistoricoTablas : BOOL
VAR_INPUT
END_VAR
// Recorre todas las lineas de la tabla una posición y añade la nueva tabla en la linea 0 para mayor coodidad al visulizar

FOR PointerHistTablas := 100 TO 1 BY -1 DO 
	RegistroLocalDataBase.aHistoricStrTablasCH2[PointerHistTablas].ID := RegistroLocalDataBase.aHistoricStrTablasCH2[PointerHistTablas-1].ID;
	RegistroLocalDataBase.aHistoricStrTablasCH2[PointerHistTablas].Fecha := RegistroLocalDataBase.aHistoricStrTablasCH2[PointerHistTablas-1].Fecha;
	RegistroLocalDataBase.aHistoricStrTablasCH2[PointerHistTablas].Modelo := RegistroLocalDataBase.aHistoricStrTablasCH2[PointerHistTablas-1].Modelo;
	RegistroLocalDataBase.aHistoricStrTablasCH2[PointerHistTablas].Formato := RegistroLocalDataBase.aHistoricStrTablasCH2[PointerHistTablas-1].Formato;
	RegistroLocalDataBase.aHistoricStrTablasCH2[PointerHistTablas].Espesor :=RegistroLocalDataBase.aHistoricStrTablasCH2[PointerHistTablas-1].Espesor;
	RegistroLocalDataBase.aHistoricStrTablasCH2[PointerHistTablas].Maquina := RegistroLocalDataBase.aHistoricStrTablasCH2[PointerHistTablas-1].Maquina;
	RegistroLocalDataBase.aHistoricStrTablasCH2[PointerHistTablas].Cont_Piezas := RegistroLocalDataBase.aHistoricStrTablasCH2[PointerHistTablas-1].Cont_Piezas;
	RegistroLocalDataBase.aHistoricStrTablasCH2[PointerHistTablas].t_Entre_Piez_Ftc := RegistroLocalDataBase.aHistoricStrTablasCH2[PointerHistTablas-1].t_Entre_Piez_Ftc;
	RegistroLocalDataBase.aHistoricStrTablasCH2[PointerHistTablas].S_Justi_Paro_Ftc := RegistroLocalDataBase.aHistoricStrTablasCH2[PointerHistTablas-1].S_Justi_Paro_Ftc;
	
END_FOR
//Estructura de la array de la tabla para visualizar el historico de la tablas pasadas
RegistroLocalDataBase.aHistoricStrTablasCH2[0].ID := PointerHistTablas;
RegistroLocalDataBase.aHistoricStrTablasCH2[0].Fecha := Fecha_PLC.StringDateHourMin;
RegistroLocalDataBase.aHistoricStrTablasCH2[0].Modelo := FuncParoNodoRemote1CorteH2.sModeloActualTabla;
RegistroLocalDataBase.aHistoricStrTablasCH2[0].Formato := FuncParoNodoRemote1CorteH2.sFormatoActualTabla;
RegistroLocalDataBase.aHistoricStrTablasCH2[0].Espesor :=FuncParoNodoRemote1CorteH2.sEspesorActualTabla;
RegistroLocalDataBase.aHistoricStrTablasCH2[0].Maquina := 'Corte húmedo 2';
RegistroLocalDataBase.aHistoricStrTablasCH2[0].Cont_Piezas := FuncParoNodoRemote1CorteH2.Funci_CortHum2.Cont_Piezas_Ftc;
RegistroLocalDataBase.aHistoricStrTablasCH2[0].t_Entre_Piez_Ftc := FuncParoNodoRemote1CorteH2.Funci_CortHum2.t_Entre_Piez_Ftc;
RegistroLocalDataBase.aHistoricStrTablasCH2[0].S_Justi_Paro_Ftc := FuncParoNodoRemote1CorteH2.Funci_CortHum2.S_Justi_Paro_Ftc;
END_METHOD

METHOD Fin_Produccion : BOOL
VAR_INPUT	
END_VAR
var
	Puls_Fin_Produccion:BOOL;	
END_VAR
//Valores por defecto del modelo y fecha de inicio modelo

s_ModeloActualTabla:= 'Sin modelo de pieza';
s_ModeloEleccionTabla:= 'Sin modelo de pieza';
s_FormatoActualTabla:= 'Sin modelo de pieza';
s_FormatoEleccionTabla:= 'Sin modelo de pieza';
s_EspesorActualTabla:= 'Sin modelo de pieza';
s_EspesorEleccionTabla:= 'Sin modelo de pieza';
s_FechaInicModeloTab:= 'Sin modelo de pieza';
 
//Reset contador de piezas 
FuncParoNodoRemote1CorteH2.Funci_CortHum2.Fin_Produccion();
END_METHOD

METHOD Inicio_Nuevo_Modelo : BOOL
VAR_INPUT
END_VAR
VAR
END_VAR

// Envías la fecha de inicio modelo de tabla 
s_FechaInicModeloTab:=Fecha_PLC.Mes_Dia_Hora_Min_Real;

//Envías el modelo de la tabla de la variable preelección  
s_ModeloActualTabla:=s_ModeloEleccionTabla;
s_FormatoActualTabla:=s_FormatoEleccionTabla;
s_EspesorActualTabla:= s_EspesorEleccionTabla;
END_METHOD

METHOD ListadoEspesorTabla : BOOL
VAR_INPUT
END_VAR
// Función para poder realizar el desplegable de espesor de la tabla en el Visu
IF IndexListEspesorTabla <> 5 THEN 
	IF IndexListEspesorTabla = 1 THEN 
		s_EspesorEleccionTabla:='3';
	END_IF
	IF IndexListEspesorTabla = 2 THEN 
		s_EspesorEleccionTabla:='6';
	END_IF
	IF IndexListEspesorTabla = 3 THEN 
		s_EspesorEleccionTabla:='12';
	END_IF
	IF IndexListEspesorTabla = 4 THEN 
		s_EspesorEleccionTabla:='20';
	END_IF
END_IF
END_METHOD

METHOD ListadoJustificacionParo : BOOL
VAR_INPUT
END_VAR
// Envío Justificación de los paros prefijados

(*Listado:  0:Sin asignar
			1: Descanso
			2: Avería
			3: Cambio de discos 
			4: Cambio de formato
			5: Cambio caballete/bandeja 
			6: Mantenimiento
			7: Falta material 
			8: Preparación material 
			9: Limpieza fin de turno 
			10: Ninguno de la lista			 
*)
//Descanso
IF IndexJustificacionParo = 1 THEN 
	FuncParoNodoRemote1CorteH2.s_JustifParoCH2 := 'Descanso';
END_IF
// Avería 
IF IndexJustificacionParo = 2 THEN 
	FuncParoNodoRemote1CorteH2.s_JustifParoCH2 := 'Avería';
END_IF
//Cambio de discos 
IF IndexJustificacionParo = 3 THEN 
	FuncParoNodoRemote1CorteH2.s_JustifParoCH2 := 'Cambio de discos';
END_IF
// Cambio de formato
IF IndexJustificacionParo = 4 THEN 
	FuncParoNodoRemote1CorteH2.s_JustifParoCH2 := 'Cambio de formato';
END_IF
//Cambio caballete/bandeja
IF IndexJustificacionParo = 5 THEN 
	FuncParoNodoRemote1CorteH2.s_JustifParoCH2 := 'Cambio caballete/bandeja';
END_IF
// Mantenimiento
IF IndexJustificacionParo = 6 THEN 
	FuncParoNodoRemote1CorteH2.s_JustifParoCH2 := 'Mantenimiento';
END_IF
// Falta de material 
IF IndexJustificacionParo = 7 THEN 
	FuncParoNodoRemote1CorteH2.s_JustifParoCH2 := 'Falta de material';
END_IF
//Preparación de material 
IF IndexJustificacionParo = 8 THEN 
	FuncParoNodoRemote1CorteH2.s_JustifParoCH2 := 'Preparación de material';
END_IF
// Limpieza fin de turno
IF IndexJustificacionParo = 9 THEN 
	FuncParoNodoRemote1CorteH2.s_JustifParoCH2 := 'Limpieza fin de turno';
END_IF
// No está en la lista
IF IndexJustificacionParo = 10 THEN 
	FuncParoNodoRemote1CorteH2.s_JustifParoCH2 := 'ESCRIBE AQUÍ LA JUSTIFICACIÓN DEL PARO';
END_IF
END_METHOD

METHOD ListFormatoTabla : BOOL
VAR_INPUT
END_VAR
// Función para poder realizar el desplegable de formato de la tabla en el Visu
IF IndexListFormatoTabla <> 8 THEN 
	IF IndexListFormatoTabla = 1 THEN 
		s_FormatoEleccionTabla:='3200 X 1500';
		Cont1:=Cont1+1;
	END_IF
	IF IndexListFormatoTabla = 2 THEN 
		s_FormatoEleccionTabla:='3600 X 1200';
		Cont2:=Cont2+1;
	END_IF
	IF IndexListFormatoTabla = 3 THEN 
		s_FormatoEleccionTabla:='1800 X 1200';
	END_IF
	IF IndexListFormatoTabla = 4 THEN 
		s_FormatoEleccionTabla:='3000 X 1000';
	END_IF
	IF IndexListFormatoTabla = 5 THEN 
		s_FormatoEleccionTabla:='2600 X 1500';
	END_IF
	IF IndexListFormatoTabla = 6 THEN 
		s_FormatoEleccionTabla:='800 X 700';
	END_IF
	IF IndexListFormatoTabla = 7 THEN 
		s_FormatoEleccionTabla:='2700 X 1000';
	END_IF
END_IF
END_METHOD

END_FUNCTION_BLOCK

// ---- POUs/Lectura_a_PLC_Maestro/Lectura_Maestro.TcPOU
PROGRAM Lectura_Maestro
VAR
	// >>>>>>>>>>>>>>>>>>>>>>>>>>>>>>>>>>>>>>>>   Estructuras de configuración con la comunicación desde y hacia el PLC Maestro <<<<<<<<<<<<<<<<<<<<<<<<<<<<<<<<<<<<<<<<<<<<<<<<<
	
	//Recordar que el IDXOFFS debe ser el doble de la posición a la que queréis acceder Ejemplo: para leer los strings a partir de la dirección MW100 Debéis poner 200 en exadecimal (C8)
	
//Configuración de la lectura de las variables Bool, IDXGRP:=16#4020(Hace referencia a la lectura de M),IDXOFFS:=16#B48C(Offset %MB46.220,  %MB46.220 a %MB46320), LEN : 101 Longitud bools leidos,DESTADDR:= ADR(Lectura_PLCs.aMasterBoolCom) Ubicación del array donde se guarda la lectura
	Config_Read_ADS_Bools_Maestro:Str_Config_ADS_to_PLC:=(NETID:='192.168.10.71.1.1', PORT:=851, IDXGRP:=16#4020,IDXOFFS:=16#B48C,LEN:=101,DESTADDR:= ADR(Lectura_PLCs.aMasterBoolCom));
	
	//Configuración de la lectura de las variables String, IDXGRP:=16#4020(Hace referencia a la lectura de M),IDXOFFS:= 16#14500(%MW42600 a %MW43815 ( 15 word)),Longitud de bytes a leer 1215 bytes = 15 strings que son 81words por cada string. ,DESTADDR:= ADR(Lectura_PLCs.aMasterStringCom) Ubicación del array donde se guarda la lectura
	Config_Read_ADS_Strings_Maestro:Str_Config_ADS_to_PLC:=(NETID:='192.168.10.71.1.1', PORT:=851, IDXGRP:=16#4020,IDXOFFS:=16#14500,LEN:=1215,DESTADDR:= ADR(Lectura_PLCs.aMasterStringCom));
	
	//Configuración de la lectura de las variables Times, IDXGRP:=16#4020(Hace referencia a la lectura de M),IDXOFFS:=16#17278 ( %MW47420 a %MW47614 (204 word),LEN:= 204 Longitud de bytes a leer bytes = 200words    51 componentes,DESTADDR:= ADR(Lectura_PLCs.aMasterTimeCom) Ubicación del array donde se guarda la lectura
	Config_Read_ADS_Times_Maestro:Str_Config_ADS_to_PLC:=(NETID:='192.168.10.71.1.1', PORT:=851, IDXGRP:=16#4020,IDXOFFS:=16#17278,LEN:= 204,DESTADDR:= ADR(Lectura_PLCs.aMasterTimeCom));
	
	//Configuración de la lectura de las variables Words, IDXGRP:=16#4020(Hace referencia a la lectura de M),IDXOFFS:=16#16008 ( %MW45060 a %MW45100 (40 word),82;//Longitud de bytes a leer 80 bytes = 40words   ,DESTADDR:= ADR(Lectura_PLCs.aMasteWordCom) Ubicación del array donde se guarda la lectura
	Config_Read_ADS_Words_Maestro:Str_Config_ADS_to_PLC:=(NETID:='192.168.10.71.1.1', PORT:=851, IDXGRP:=16#4020,IDXOFFS:=16#16008,LEN:=82,DESTADDR:= ADR(Lectura_PLCs.aMasterWordCom));
	
	fbLectura_a_PLC_Maestro:fbLectura_a_PLC;
	

END_VAR
VAR_INPUT
	bNextBlockToRead_L4_Done:BOOL;
END_VAR

fbLectura_a_PLC_Maestro(
	Config_PLC_ADS_Bools:=Config_Read_ADS_Bools_Maestro,
	Config_PLC_ADS_Strings:=Config_Read_ADS_Strings_Maestro,
	Config_PLC_ADS_Times:=Config_Read_ADS_Times_Maestro,
	Config_PLC_ADS_Words:=Config_Read_ADS_Words_Maestro,
 	TimeReadStateEntreLecturas:=T#20MS,
	bHabilitadaLectura:=TRUE,
	);

END_PROGRAM

// ---- GlobalTextList.TcGTLO
TEXTLIST GlobalTextList
  505 = '%i'
  650 = '%s'
  177 = '%s \tContador piezas corte húmedo 4 '
  771 = '%s \tContador piezas Multidiscos 2'
  56 = "%t[H'h'm'min']"
  702 = '%t[HH,mm]'
  1013 = '%t[HH:mm]h'
  410 = '%t[HHmm]'
  696 = '%t[H]h[m]min'
  175 = '%t[min]'
  633 = '%t[s,ms]'
  1163 = 'ACEPTAR'
  1790 = 'AJUSTE\nMEDIDAS/PRECORTE'
  152 = 'Ajustes'
  636 = 'Atrás'
  589 = 'AVERÍA'
  1710 = 'CAMBIO \nCABALLETE/BANDEJA'
  1137 = 'CAMBIO DISCOS'
  288 = 'CAMBIO FORMATO'
  856 = 'Contador de piezas'
  115 = 'Corte húmedo 2'
  548 = 'CORTE HÚMEDO 2'
  979 = 'Corte húmedo 3'
  913 = 'CORTE HÚMEDO 3'
  137 = 'Corte húmedo 4'
  1186 = 'CORTE HÚMEDO 4'
  952 = 'Decoración'
  448 = 'Delay Escritura'
  1310 = 'DESCANSO'
  503 = 'Diagnóstico lineas'
  1366 = 'Día'
  765 = 'Elige la línea la cual quieres ver el estado de sus contadores y señales'
  630 = 'En producción'
  432 = 'En producción todo OK'
  331 = 'En produccoón desde:    %s'
  434 = 'Entrada Horno Inferior '
  370 = 'Entrada Horno Superior'
  557 = 'Entrada secadero'
  466 = 'Entre Piez %s'
  850 = 'Entre Piez Anterior %s'
  740 = 'ESPESOR'
  631 = 'Espesor'
  818 = 'Exit'
  1436 = 'FALTA DE MATERIAL'
  1029 = 'Fecha'
  394 = 'Fecha inicio del modelo actual'
  297 = 'Filtro Down'
  866 = 'Filtro Up'
  796 = 'Fin de producción del modelo'
  766 = 'FINALIZAR MODELO'
  79 = 'FORMATO'
  419 = 'Formato'
  884 = 'Forzar Fotocelula'
  768 = 'Habilitar escritura \nen MySQL'
  350 = 'Habilitar escritura Linea 4\nen MySQL'
  841 = 'Habilitar lectura a\nPLC L4'
  332 = 'Habilitar lectura a\nPLCs'
  34 = 'Habilitar lectura al\nPLC Maestro'
  907 = 'HISTÓRICO'
  532 = 'Histórico'
  248 = 'HISTÓRICO PRODUCCIÓN'
  689 = 'Home'
  681 = 'Hora Fin Paro'
  1204 = 'HORA INICIO'
  553 = 'Hora Inicio del paro'
  340 = 'Hora Inicio Paro'
  358 = 'Horno Inf.'
  962 = 'Horno Sup.'
  733 = 'ID'
  867 = 'INICIADA:'
  798 = 'Inicio'
  1088 = 'INICIO'
  1183 = 'Justif paro'
  895 = 'Justificación del paro'
  266 = 'JUSTIFICAR EL PARO ACTUAL'
  1063 = 'JUSTIFICAR PARO'
  39 = 'LIMPIEZA FIN DE TURNO'
  67 = 'Línea en paro'
  1024 = 'MANTENIMIENTO'
  596 = 'Maquina'
  227 = 'Marca Paro '
  911 = 'Marca Sin Paro '
  316 = 'Min'
  914 = 'Minutos Parado'
  1198 = 'MODELO'
  531 = 'Modelo'
  735 = 'Modelo actual'
  659 = 'Modelo:'
  873 = 'MOTIVO 1'
  228 = 'Multidiscos 1'
  197 = 'MULTIDISCOS 1'
  118 = 'Multidiscos 2'
  989 = 'MULTIDISCOS 2'
  1014 = 'NINGÚN PARO ACTIVO'
  615 = 'NO ESTÁ EN LA LISTA'
  1148 = 'NUEVO MODELO'
  145 = 'Numero de tablas'
  1060 = 'Número de losas'
  490 = 'Paro activo'
  1136 = 'PARO ACTIVO'
  1107 = 'PARO ACTUAL'
  1678 = 'PARO TOTAL ACUMULADO '
  566 = 'PAROS'
  21 = 'PARÁMETROS'
  1311 = 'PIEZAS'
  329 = 'Prensa'
  307 = 'PREPARACION MATERIAL'
  935 = 'PRODUCCIÓN'
  258 = 'PRODUCIDAS'
  600 = 'Página de diagnóstico'
  732 = 'Reset contador'
  1413 = 'Revisa que no haya ninguna pieza en la línea.'
  463 = 'Salida Airless 2'
  618 = 'Salida Greencut'
  193 = 'Secadero'
  403 = 'Seg'
  225 = 'Sensor presencia tabla '
  906 = 'Tiempo entre Piezas'
  64 = 'tiempo entre Piezas'
  55 = 'Tiempo entre Piezas\nAnterior'
  774 = 'Tiempo entre tablas'
  649 = 'Tiempo filtrado fotocelulas\npara evitar parpadeos'
  501 = 'Tiempo para empezar \na contar como paro'
  433 = 'Total piezas'
  997 = 'Turno'
  173 = 'TURNO ACTUAL'
  123 = 'Ultima Frase enviada a MySQL '
  1166 = 'VOLVER'
  1577 = '¿Quieres finalizar el modelo?'
END_TEXTLIST

// ---- VISUs/Ajustes_CorteH2.TcVIS
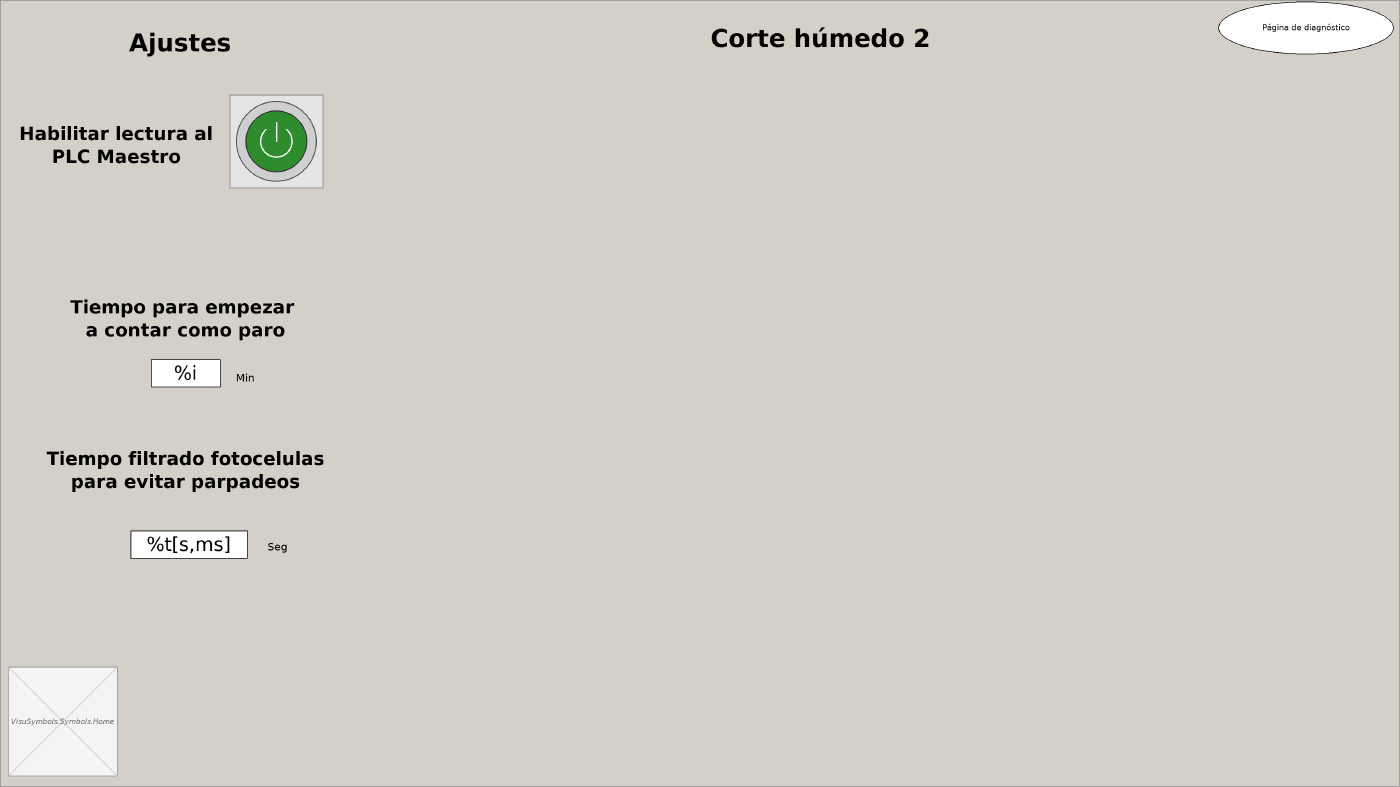
VISUALIZATION Ajustes_CorteH2  // 1920x1080
    Label (143,29 208x59), "Ajustes"
    Image (11,915 150x150), image: VisuSymbols.Symbols.Home
        OnMouseClick: change screen: Home_CortH2
    Label (22,144 275x110), "Habilitar lectura al PLC Maestro"
    PowerSwitch (315,128 128x132), variable: MAIN_Orden_Lectura_PLCs.bHabilitaLectura_Maestro, behaviour: TOGGLE, style: Switch-PowerSwitch-Green
    Label (82,390 345x94), "Tiempo para empezar a contar como paro"
    Label (160,482 188x30)
    Rectangle (207,493 95x38), "%i", text variable: FuncParoNodoRemote1CorteH2.HMI_Tiempo_Offset_MParo
        OnMouseDown: write the text variable via Edit
    Label (307,500 59x37), "Min"
    Label (58,598 393x94), "Tiempo filtrado fotocelulas para evitar parpadeos"
    Label (351,732 59x37), "Seg"
    Rectangle (179,728 160x38), "%t[s,ms]", text variable: FuncParoNodoRemote1CorteH2.HMI_TiempoFiltradoFotocel
        OnMouseDown: write the text variable via Edit
    Label (925,23 401x59), "Corte húmedo 2"
    Ellipse (1671,2 240x72), "Página de diagnóstico"
        OnMouseClick: change screen: DiagnosticoFB
END_VISUALIZATION

// ---- VISUs/Ajustes_CorteH3.TcVIS
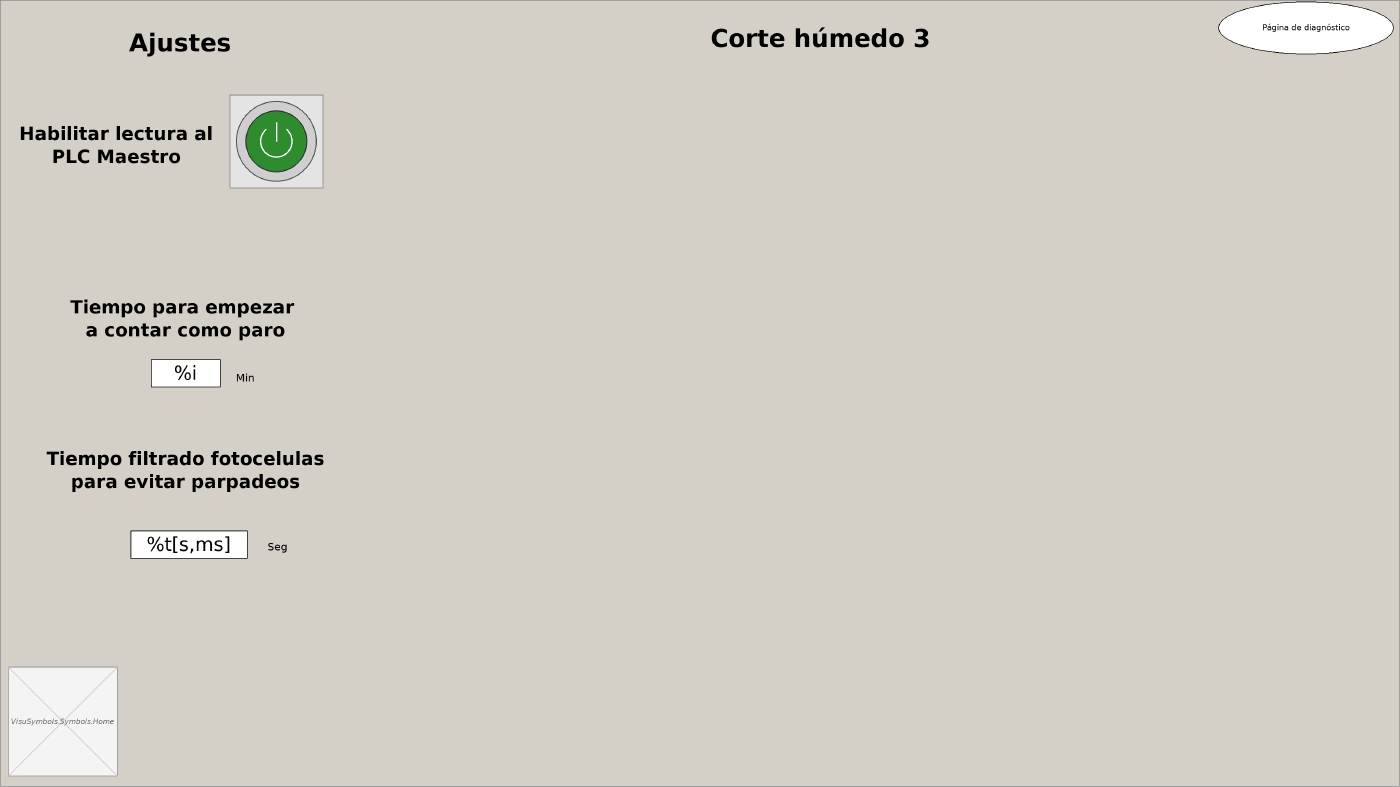
VISUALIZATION Ajustes_CorteH3  // 1920x1080
    Label (143,29 208x59), "Ajustes"
    Image (11,915 150x150), image: VisuSymbols.Symbols.Home
        OnMouseClick: change screen: Home_CortH2
    Label (22,144 275x110), "Habilitar lectura al PLC Maestro"
    PowerSwitch (315,128 128x132), variable: MAIN_Orden_Lectura_PLCs.bHabilitaLectura_Maestro, behaviour: TOGGLE, style: Switch-PowerSwitch-Green
    Label (82,390 345x94), "Tiempo para empezar a contar como paro"
    Label (160,482 188x30)
    Rectangle (207,493 95x38), "%i", text variable: FuncParoNodoLocalCorteH3.HMI_Tiempo_Offset_MParo
        OnMouseDown: write the text variable via Edit
    Label (307,500 59x37), "Min"
    Label (58,598 393x94), "Tiempo filtrado fotocelulas para evitar parpadeos"
    Label (351,732 59x37), "Seg"
    Rectangle (179,728 160x38), "%t[s,ms]", text variable: FuncParoNodoLocalCorteH3.HMI_TiempoFiltradoFotocel
        OnMouseDown: write the text variable via Edit
    Label (925,23 401x59), "Corte húmedo 3"
    Ellipse (1671,2 240x72), "Página de diagnóstico"
        OnMouseClick: change screen: DiagnosticoFB
END_VISUALIZATION

// ---- VISUs/DiagnosticoFB.TcVIS
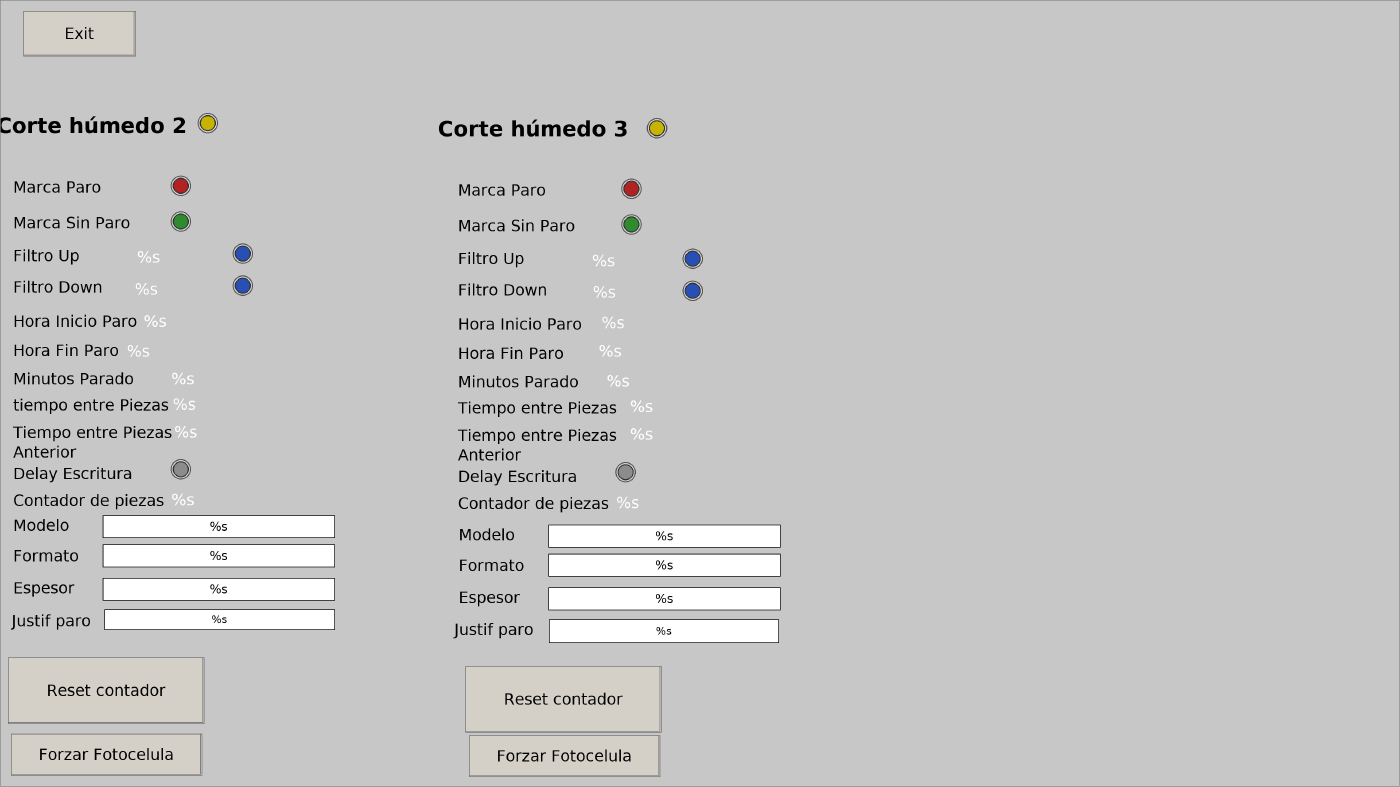
VISUALIZATION DiagnosticoFB  // 1920x1080
    Rectangle (185,338 93x30), "%s", text variable: FuncParoNodoRemote1CorteH2.Funci_CortHum2.tFiltro_up_Ftc.ET
    Label (10,146 231x53), "Corte húmedo 2"
    Label (15,242 150x30), "Marca Paro"
    Lamp1 (269,153 32x32), variable: FuncParoNodoRemote1CorteH2.Funci_CortHum2.Fotocelula, style: Lamp-Lamp1-Yellow
    Lamp1 (232,239 32x32), variable: FuncParoNodoRemote1CorteH2.Funci_CortHum2.MParo_Ftc, style: Lamp-Lamp1-Red
    Label (15,291 188x30), "Marca Sin Paro"
    Lamp1 (232,288 32x32), variable: FuncParoNodoRemote1CorteH2.Funci_CortHum2.M_SinParo_Ftc, style: Lamp-Lamp1-Green
    Label (15,336 117x30), "Filtro Up"
    Rectangle (182,382 93x30), "%s", text variable: FuncParoNodoRemote1CorteH2.Funci_CortHum2.tFiltro_down_Ftc.ET
    Label (15,379 143x30), "Filtro Down"
    Rectangle (194,426 183x30), "%s", text variable: FuncParoNodoRemote1CorteH2.Funci_CortHum2.H_InParo_Ftc
    Label (15,426 204x30), "Hora Inicio Paro"
    Lamp1 (317,332 32x32), variable: FuncParoNodoRemote1CorteH2.Funci_CortHum2.tFiltro_up_Ftc.Q, style: Lamp-Lamp1-Blue
    Lamp1 (317,376 32x32), variable: FuncParoNodoRemote1CorteH2.Funci_CortHum2.tFiltro_down_Ftc.Q, style: Lamp-Lamp1-Blue
    Rectangle (171,467 179x30), "%s", text variable: FuncParoNodoRemote1CorteH2.Funci_CortHum2.H_FinParo_Ftc
    Label (15,466 204x30), "Hora Fin Paro"
    Rectangle (232,505 192x30), "%s", text variable: FuncParoNodoRemote1CorteH2.Funci_CortHum2.Min_Parado_Ftc
    Label (15,505 204x30), "Minutos Parado"
    Label (15,541 244x30), "tiempo entre Piezas"
    Label (15,576 255x62), "Tiempo entre Piezas Anterior"
    Label (15,635 204x30), "Delay Escritura"
    Rectangle (232,671 93x30), "%s", text variable: FuncParoNodoRemote1CorteH2.Funci_CortHum2.Cont_Piezas_Ftc
    Label (15,672 215x30), "Contador de piezas"
    Lamp1 (232,628 32x32), variable: FuncParoNodoRemote1CorteH2.Funci_CortHum2.Delay_Esc_Ftc.Q, style: Lamp-Lamp1-Gray
    Button (32,15 154x62), "Exit"
        OnMouseClick: change screen: Home_CortH2
    Rectangle (809,343 93x30), "%s", text variable: FuncParoNodoLocalCorteH3.Funci_CortHum3.tFiltro_up_Ftc.ET
    Label (599,134 264x86), "Corte húmedo 3"
    Label (625,246 150x30), "Marca Paro"
    Lamp1 (885,160 32x32), variable: FuncParoNodoLocalCorteH3.Funci_CortHum3.Fotocelula, style: Lamp-Lamp1-Yellow
    Lamp1 (850,243 32x32), variable: FuncParoNodoLocalCorteH3.Funci_CortHum3.MParo_Ftc, style: Lamp-Lamp1-Red
    Label (625,295 188x30), "Marca Sin Paro"
    Lamp1 (850,292 32x32), variable: FuncParoNodoLocalCorteH3.Funci_CortHum3.M_SinParo_Ftc, style: Lamp-Lamp1-Green
    Label (625,340 117x30), "Filtro Up"
    Rectangle (810,386 93x30), "%s", text variable: FuncParoNodoLocalCorteH3.Funci_CortHum3.tFiltro_down_Ftc.ET
    Label (625,383 143x30), "Filtro Down"
    Rectangle (822,428 183x30), "%s", text variable: FuncParoNodoLocalCorteH3.Funci_CortHum3.H_InParo_Ftc
    Label (625,430 204x30), "Hora Inicio Paro"
    Lamp1 (934,339 32x32), variable: FuncParoNodoLocalCorteH3.Funci_CortHum3.tFiltro_up_Ftc.Q, style: Lamp-Lamp1-Blue
    Lamp1 (934,383 32x32), variable: FuncParoNodoLocalCorteH3.Funci_CortHum3.tFiltro_down_Ftc.Q, style: Lamp-Lamp1-Blue
    Rectangle (818,467 179x30), "%s", text variable: FuncParoNodoLocalCorteH3.Funci_CortHum3.H_FinParo_Ftc
    Label (625,470 204x30), "Hora Fin Paro"
    Rectangle (829,508 192x30), "%s", text variable: FuncParoNodoLocalCorteH3.Funci_CortHum3.Min_Parado_Ftc
    Label (625,509 204x30), "Minutos Parado"
    Label (625,545 244x30), "Tiempo entre Piezas"
    Label (625,580 255x62), "Tiempo entre Piezas Anterior"
    Label (625,639 204x30), "Delay Escritura"
    Rectangle (842,675 93x30), "%s", text variable: FuncParoNodoLocalCorteH3.Funci_CortHum3.Cont_Piezas_Ftc
    Label (625,676 215x30), "Contador de piezas"
    Lamp1 (842,632 32x32), variable: FuncParoNodoLocalCorteH3.Funci_CortHum3.Delay_Esc_Ftc.Q, style: Lamp-Lamp1-Gray
    Rectangle (234,540 192x30), "%s", text variable: FuncParoNodoRemote1CorteH2.Funci_CortHum2.t_Entre_Piez_Ftc
    Rectangle (861,543 192x30), "%s", text variable: FuncParoNodoLocalCorteH3.Funci_CortHum3.t_Entre_Piez_Ftc
    Rectangle (236,578 192x30), "%s", text variable: FuncParoNodoRemote1CorteH2.Funci_CortHum2.t_Entr_Piez_Ante_Ftc
    Rectangle (861,581 192x30), "%s", text variable: FuncParoNodoLocalCorteH3.Funci_CortHum3.t_Entr_Piez_Ante_Ftc
    Button (11,902 269x91), "Reset contador"
        tap FuncParoNodoRemote1CorteH2.Funci_CortHum2.ResetContPiez
    Button (638,914 269x91), "Reset contador"
        tap FuncParoNodoLocalCorteH3.Funci_CortHum3.ResetContPiez
    Button (643,1009 262x57), "Forzar Fotocelula"
        tap FuncParoNodoLocalCorteH3.ForzadoFtcCortHum3
    Button (15,1007 262x57), "Forzar Fotocelula"
        tap FuncParoNodoRemote1CorteH2.ForzadoFtcCortHum2
    Label (15,706 92x30), "Modelo"
    Label (15,748 105x30), "Formato"
    Label (15,792 99x30), "Espesor"
    Rectangle (141,707 318x31), "%s", text variable: FuncParoNodoRemote1CorteH2.FunGeneCortHum2.s_ModeloActualTabla
        OnMouseDown: write the text variable via Edit
    Rectangle (141,747 318x31), "%s", text variable: FuncParoNodoRemote1CorteH2.FunGeneCortHum2.s_FormatoActualTabla
        OnMouseDown: write the text variable via Edit
    Rectangle (141,793 318x31), "%s", text variable: FuncParoNodoRemote1CorteH2.FunGeneCortHum2.s_EspesorActualTabla
        OnMouseDown: write the text variable via Edit
    Label (626,719 92x30), "Modelo"
    Label (626,761 105x30), "Formato"
    Label (626,805 99x30), "Espesor"
    Rectangle (752,720 318x31), "%s", text variable: FuncParoNodoLocalCorteH3.FunGeneCortHum3.s_ModeloActualTabla
        OnMouseDown: write the text variable via Edit
    Rectangle (752,760 318x31), "%s", text variable: FuncParoNodoLocalCorteH3.FunGeneCortHum3.s_FormatoActualTabla
        OnMouseDown: write the text variable via Edit
    Rectangle (752,806 318x31), "%s", text variable: FuncParoNodoLocalCorteH3.FunGeneCortHum3.s_EspesorActualTabla
        OnMouseDown: write the text variable via Edit
    Label (13,837 123x30), "Justif paro"
    Rectangle (143,836 316x28), "%s", text variable: FuncParoNodoRemote1CorteH2.Funci_CortHum2.S_Justi_Paro_Ftc
        OnMouseDown: write the text variable via Edit
    Rectangle (753,850 315x32), "%s", text variable: FuncParoNodoLocalCorteH3.Funci_CortHum3.S_Justi_Paro_Ftc
        OnMouseDown: write the text variable via Edit
    Label (620,849 123x30), "Justif paro"
END_VISUALIZATION

// ---- VISUs/HistTablaTablas_Ch2.TcVIS
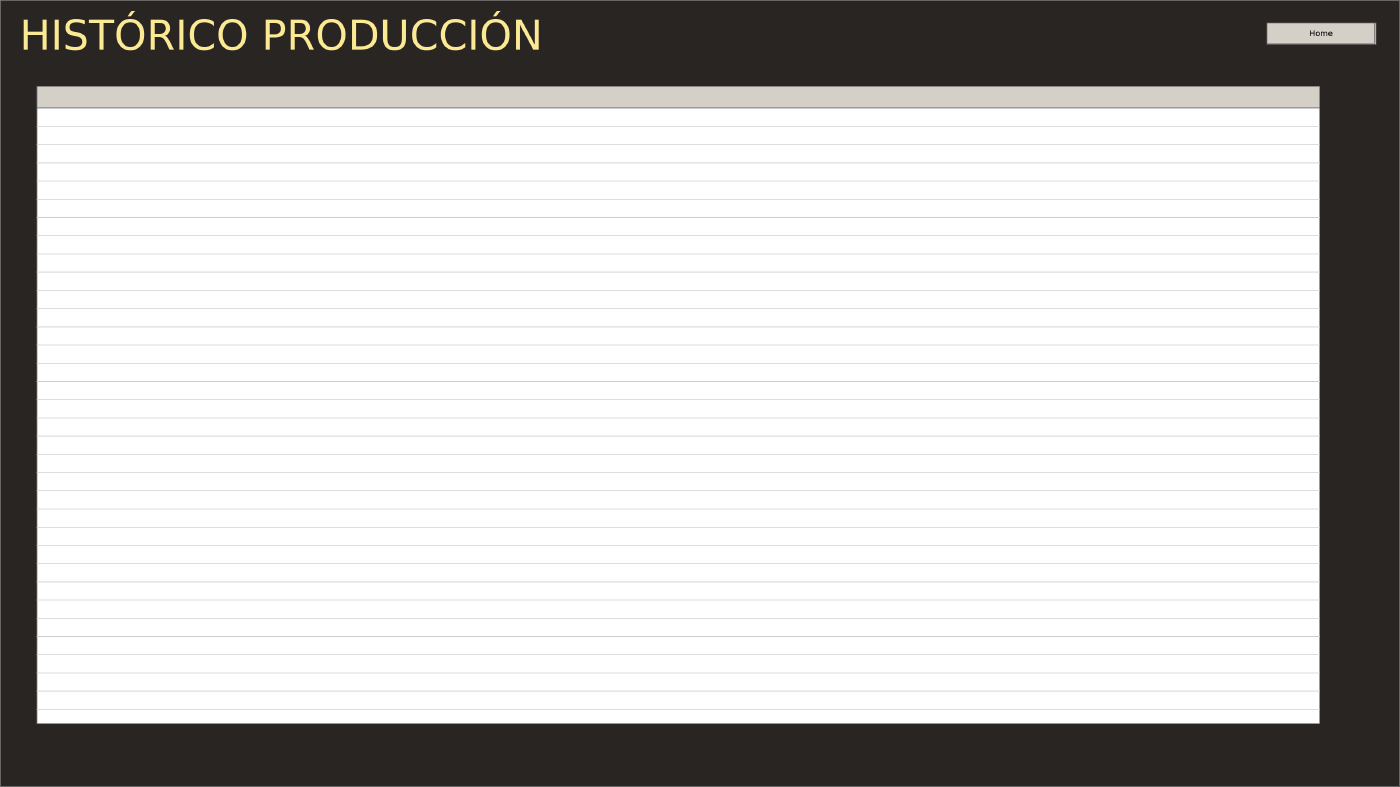
VISUALIZATION HistTablaTablas_Ch2  // 1920x1080
    Table (50,118 1760x875), data array: RegistroLocalDataBase.aHistoricStrTablasCH2
        p3854506369: RegistroLocalDataBase.aHistoricStrTablasCH2[INDEX].ID
        p1892666644: RegistroLocalDataBase.aHistoricStrTablasCH2[INDEX].Fecha
        p338671338: RegistroLocalDataBase.aHistoricStrTablasCH2[INDEX].Modelo
        p2170511999: RegistroLocalDataBase.aHistoricStrTablasCH2[INDEX].Formato
        p3723444502: RegistroLocalDataBase.aHistoricStrTablasCH2[INDEX].Espesor
        p1218418051: RegistroLocalDataBase.aHistoricStrTablasCH2[INDEX].Maquina
        p746581629: RegistroLocalDataBase.aHistoricStrTablasCH2[INDEX].Cont_Piezas
        p3104783080: RegistroLocalDataBase.aHistoricStrTablasCH2[INDEX].t_Entre_Piez_Ftc
        p2501879983: RegistroLocalDataBase.aHistoricStrTablasCH2[INDEX].S_Justi_Paro_Ftc
        p1757482276: Numero de tablas
        p4088588272: Tiempo entre tablas
        p2243050616: Justificación del paro
    Label (24,16 669x64), "HISTÓRICO PRODUCCIÓN"
    Button (1737,31 150x30), "Home"
        OnMouseClick: change screen: Home_CortH2
END_VISUALIZATION

// ---- VISUs/HistTablaTablas_Ch3.TcVIS
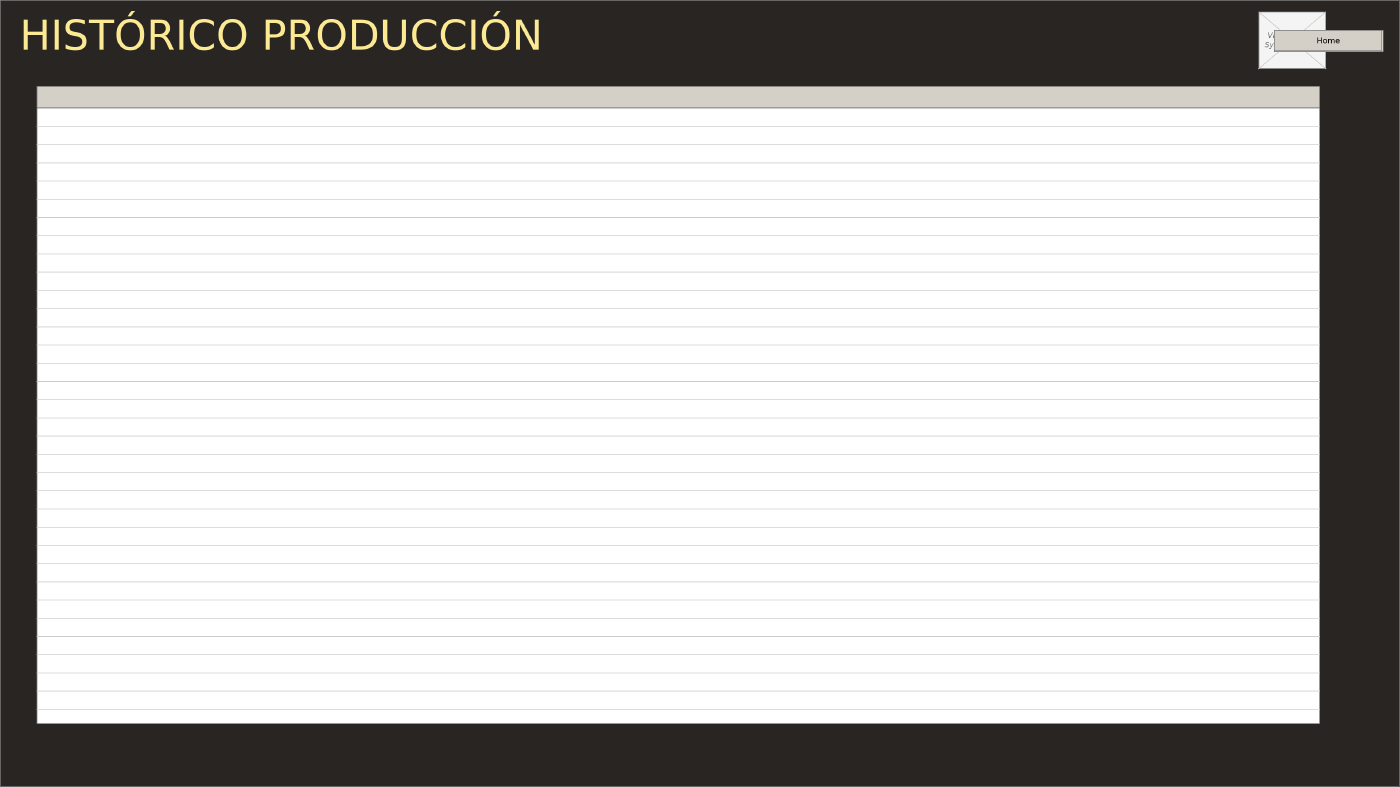
VISUALIZATION HistTablaTablas_Ch3  // 1920x1080
    Image (1726,16 92x78), image: VisuSymbols.Symbols.Home
        OnMouseClick: change screen: Home_CortH2
    Table (50,118 1760x875), data array: RegistroLocalDataBase.aHistoricStrTablasCH3
        p3854506369: RegistroLocalDataBase.aHistoricStrTablasCH3[INDEX].ID
        p1892666644: RegistroLocalDataBase.aHistoricStrTablasCH3[INDEX].Fecha
        p338671338: RegistroLocalDataBase.aHistoricStrTablasCH3[INDEX].Modelo
        p2170511999: RegistroLocalDataBase.aHistoricStrTablasCH3[INDEX].Formato
        p3723444502: RegistroLocalDataBase.aHistoricStrTablasCH3[INDEX].Espesor
        p1218418051: RegistroLocalDataBase.aHistoricStrTablasCH3[INDEX].Maquina
        p746581629: RegistroLocalDataBase.aHistoricStrTablasCH3[INDEX].Cont_Piezas
        p3104783080: RegistroLocalDataBase.aHistoricStrTablasCH3[INDEX].t_Entre_Piez_Ftc
        p2501879983: RegistroLocalDataBase.aHistoricStrTablasCH3[INDEX].S_Justi_Paro_Ftc
        p1757482276: Numero de tablas
        p4088588272: Tiempo entre tablas
        p2243050616: Justificación del paro
    Label (24,16 669x64), "HISTÓRICO PRODUCCIÓN"
    Button (1747,41 150x30), "Home"
        OnMouseClick: change screen: Home_CortH3
END_VISUALIZATION

// ---- VISUs/Home_CortH2.TcVIS
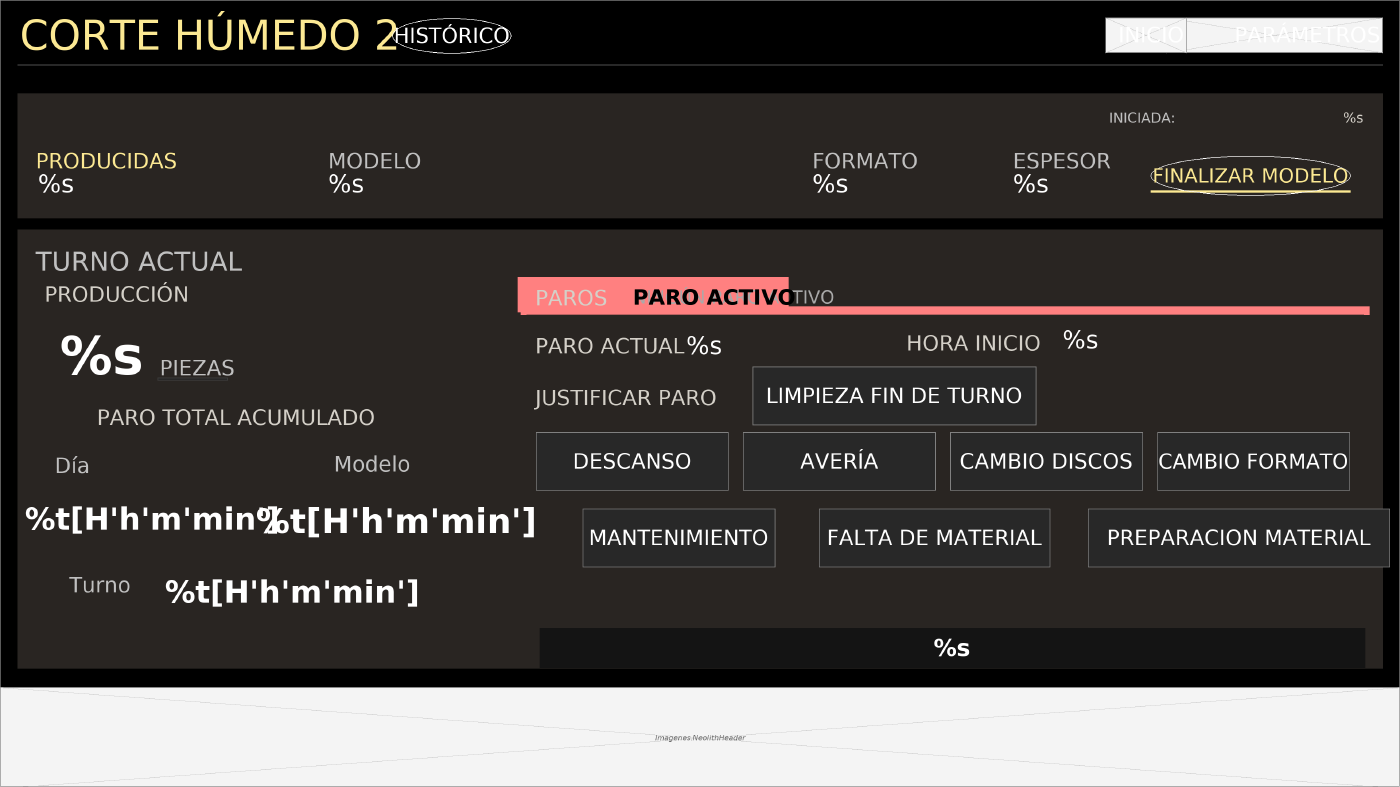
VISUALIZATION Home_CortH2  // 1920x1080
    Rectangle (24,315 1872x602)
    Rectangle (24,128 1872x171)
    Rectangle (24,88 1872x2)
    Label (24,16 514x64), "CORTE HÚMEDO 2"
    Rectangle (1454,451 375x30), "%s", text variable: FuncParoNodoRemote1CorteH2.Funci_CortHum2.H_InParo_Ftc, invisible if: FuncParoNodoRemote1CorteH2.Funci_CortHum2.M_SinParo_Ftc
    Rectangle (938,459 287x30), "%s", text variable: FuncParoNodoRemote1CorteH2.Funci_CortHum2.Min_Parado_Ftc, invisible if: FuncParoNodoRemote1CorteH2.Funci_CortHum2.M_SinParo_Ftc
    Rectangle (1573,147 300x30), "%s", text variable: FuncParoNodoRemote1CorteH2.sFechaInicModeloTab
    Label (1518,147 99x30), "INICIADA:"
    Rectangle (740,862 1132x54), "%s", text variable: FuncParoNodoRemote1CorteH2.Funci_CortHum2.S_Justi_Paro_Ftc, invisible if: FuncParoNodoRemote1CorteH2.Funci_CortHum2.M_SinParo_Ftc, input disabled if: FuncParoNodoRemote1CorteH2.FunGeneCortHum2.IndexJustificacionParo<>10
        OnMouseDown: write the text variable via Edit
    Image (1600,24 296x48), "PARÁMETROS"
        OnMouseClick: change screen: Ajustes_CorteH2
    Image (1516,24 111x48), "INICIO"
        OnMouseClick: change screen: Home_Sel_Maq
    Group (447,203 1095x69)
        Rectangle (0,29 671x40), "%s", text variable: FuncParoNodoRemote1CorteH2.sModeloActualTabla
        Rectangle (939,29 120x40), "%s", text variable: FuncParoNodoRemote1CorteH2.sEspesorActualTabla
        Rectangle (664,29 321x40), "%s", text variable: FuncParoNodoRemote1CorteH2.sFormatoActualTabla
        Label (0,0 487x36), "MODELO"
        Label (664,0 156x36), "FORMATO"
        Label (939,0 156x36), "ESPESOR"
    Label (46,203 199x36), "PRODUCIDAS"
    Rectangle (49,232 248x40), "%s", text variable: FuncParoNodoRemote1CorteH2.Funci_CortHum2.Cont_Piezas_Ftc
    Group (1578,214 274x54)
        Rectangle (0,47 274x3)
        Ellipse (0,0 274x54), "FINALIZAR MODELO"
            OnMouseClick: OpenDialog Dialog=V_Emerg_Fin_Prod_Ch2, OpenModal=True, OpenCentered=True
    Label (46,332 390x54), "TURNO ACTUAL"
    Label (58,386 199x36), "PRODUCCIÓN"
    Label (731,457 261x36), "PARO ACTUAL", invisible if: FuncParoNodoRemote1CorteH2.Funci_CortHum2.M_SinParo_Ftc
    Label (1240,453 261x36), "HORA INICIO", invisible if: FuncParoNodoRemote1CorteH2.Funci_CortHum2.M_SinParo_Ftc
    RoundedRectangle (735,593 264x80), "DESCANSO", invisible if: FuncParoNodoRemote1CorteH2.Funci_CortHum2.M_SinParo_Ftc
        OnMouseClick: execute { FuncParoNodoRemote1CorteH2.FunGeneCortHum2.IndexJustificacionParo:=1; FuncParoNodoRemote1CorteH2.FunGeneCortHum2.ListadoJustificacionParo(); }
    RoundedRectangle (1019,593 264x80), "AVERÍA", invisible if: FuncParoNodoRemote1CorteH2.Funci_CortHum2.M_SinParo_Ftc
        OnMouseClick: execute { FuncParoNodoRemote1CorteH2.FunGeneCortHum2.IndexJustificacionParo:=2; FuncParoNodoRemote1CorteH2.FunGeneCortHum2.ListadoJustificacionParo(); }
    RoundedRectangle (1303,593 264x80), "CAMBIO DISCOS", invisible if: FuncParoNodoRemote1CorteH2.Funci_CortHum2.M_SinParo_Ftc
        OnMouseClick: execute { FuncParoNodoRemote1CorteH2.FunGeneCortHum2.IndexJustificacionParo:=3; FuncParoNodoRemote1CorteH2.FunGeneCortHum2.ListadoJustificacionParo(); }
    RoundedRectangle (1587,593 264x80), "CAMBIO FORMATO", invisible if: FuncParoNodoRemote1CorteH2.Funci_CortHum2.M_SinParo_Ftc
        OnMouseClick: execute { FuncParoNodoRemote1CorteH2.FunGeneCortHum2.IndexJustificacionParo:=4; FuncParoNodoRemote1CorteH2.FunGeneCortHum2.ListadoJustificacionParo(); }
    Rectangle (79,444 183x88), "%s", text variable: FuncParoNodoRemote1CorteH2.Funci_CortHum2.Cont_Piezas_Ftc
    Label (216,487 106x36), "PIEZAS"
    Rectangle (216,518 96x4), colour toggle: FuncParoNodoRemote1CorteH2.Funci_CortHum2.Fotocelula
    Label (731,528 261x36), "JUSTIFICAR PARO", invisible if: FuncParoNodoRemote1CorteH2.Funci_CortHum2.M_SinParo_Ftc
    Rectangle (714,424 1164x4), invisible if: FuncParoNodoRemote1CorteH2.Funci_CortHum2.M_SinParo_Ftc
    Rectangle (710,380 371x48), invisible if: FuncParoNodoRemote1CorteH2.Funci_CortHum2.M_SinParo_Ftc
    Label (731,391 199x36), "PAROS", invisible if: FuncParoNodoRemote1CorteH2.Funci_CortHum2.M_SinParo_Ftc
    Label (865,393 326x30), "NINGÚN PARO ACTIVO", invisible if: FuncParoNodoRemote1CorteH2.Funci_CortHum2.MParo_Ftc
    Label (865,393 235x30), "PARO ACTIVO", invisible if: FuncParoNodoRemote1CorteH2.Funci_CortHum2.M_SinParo_Ftc
    Ellipse (538,25 163x48), "HISTÓRICO"
        OnMouseClick: change screen: HistTablaTablas_Ch2
    Label (130,555 367x36), "PARO TOTAL ACUMULADO"
    Image (-3,943 1927x139), image: Imagenes.NeolithHeader
    RoundedRectangle (799,698 264x80), "MANTENIMIENTO", invisible if: FuncParoNodoRemote1CorteH2.Funci_CortHum2.M_SinParo_Ftc
        OnMouseClick: execute { FuncParoNodoRemote1CorteH2.FunGeneCortHum2.IndexJustificacionParo:=6; FuncParoNodoRemote1CorteH2.FunGeneCortHum2.ListadoJustificacionParo(); }
    RoundedRectangle (1123,698 317x80), "FALTA DE MATERIAL", invisible if: FuncParoNodoRemote1CorteH2.Funci_CortHum2.M_SinParo_Ftc
        OnMouseClick: execute { FuncParoNodoRemote1CorteH2.FunGeneCortHum2.IndexJustificacionParo:=7; FuncParoNodoRemote1CorteH2.FunGeneCortHum2.ListadoJustificacionParo(); }
    RoundedRectangle (1492,698 414x80), "PREPARACION MATERIAL", invisible if: FuncParoNodoRemote1CorteH2.Funci_CortHum2.M_SinParo_Ftc
        OnMouseClick: execute { FuncParoNodoRemote1CorteH2.FunGeneCortHum2.IndexJustificacionParo:=8; FuncParoNodoRemote1CorteH2.FunGeneCortHum2.ListadoJustificacionParo(); }
    RoundedRectangle (1032,503 389x80), "LIMPIEZA FIN DE TURNO", invisible if: FuncParoNodoRemote1CorteH2.Funci_CortHum2.M_SinParo_Ftc
        OnMouseClick: execute { FuncParoNodoRemote1CorteH2.FunGeneCortHum2.IndexJustificacionParo:=9; FuncParoNodoRemote1CorteH2.FunGeneCortHum2.ListadoJustificacionParo(); }
    Rectangle (31,668 295x88), "%t[H'h'm'min']", text variable: FuncParoNodoRemote1CorteH2.Funci_CortHum2.fbTiempParoAcumDiario.t_Acumulado
    Label (72,621 76x36), "Día"
    Rectangle (223,768 325x88), "%t[H'h'm'min']", text variable: FuncParoNodoRemote1CorteH2.Funci_CortHum2.fbTiempParoAcumTurno.t_Acumulado
    Label (92,785 102x36), "Turno"
    Rectangle (348,671 388x88), "%t[H'h'm'min']", text variable: FuncParoNodoRemote1CorteH2.Funci_CortHum2.fbTiempParoAcumModelo.t_Acumulado
    Label (455,619 118x36), "Modelo"
END_VISUALIZATION

// ---- VISUs/Home_CortH3.TcVIS
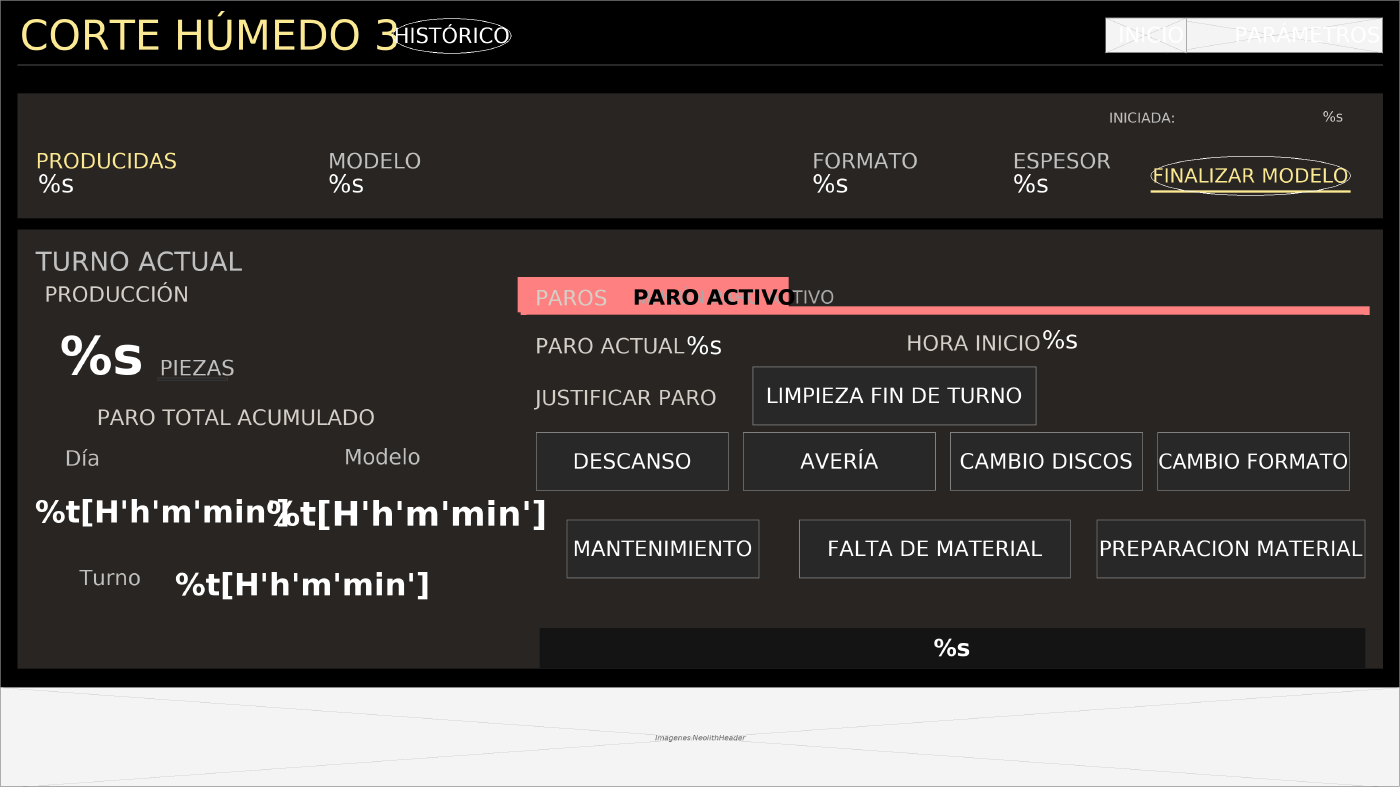
VISUALIZATION Home_CortH3  // 1920x1080
    Rectangle (24,315 1872x602)
    Rectangle (24,128 1872x171)
    Rectangle (24,88 1872x2)
    Label (24,16 514x64), "CORTE HÚMEDO 3"
    Rectangle (1426,451 183x30), "%s", text variable: FuncParoNodoLocalCorteH3.Funci_CortHum3.H_InParo_Ftc, invisible if: FuncParoNodoLocalCorteH3.Funci_CortHum3.M_SinParo_Ftc
    Rectangle (938,459 192x30), "%s", text variable: FuncParoNodoLocalCorteH3.Funci_CortHum3.Min_Parado_Ftc, invisible if: FuncParoNodoLocalCorteH3.Funci_CortHum3.M_SinParo_Ftc
    Rectangle (1573,147 272x27), "%s", text variable: FuncParoNodoLocalCorteH3.sFechaInicModeloTab
    Label (1518,147 99x30), "INICIADA:"
    Rectangle (740,862 1132x54), "%s", text variable: FuncParoNodoLocalCorteH3.Funci_CortHum3.S_Justi_Paro_Ftc, invisible if: FuncParoNodoLocalCorteH3.Funci_CortHum3.M_SinParo_Ftc, input disabled if: FuncParoNodoLocalCorteH3.FunGeneCortHum3.IndexJustificacionParo<>10
        OnMouseDown: write the text variable via Edit
    Image (1600,24 296x48), "PARÁMETROS"
        OnMouseClick: change screen: Ajustes_CorteH3
    Image (1516,24 111x48), "INICIO"
        OnMouseClick: change screen: Home_Sel_Maq
    Rectangle (447,232 671x40), "%s", text variable: FuncParoNodoLocalCorteH3.sModeloActualTabla
    Rectangle (1386,232 120x40), "%s", text variable: FuncParoNodoLocalCorteH3.FunGeneCortHum3.s_EspesorActualTabla
    Rectangle (1111,232 275x40), "%s", text variable: FuncParoNodoLocalCorteH3.FunGeneCortHum3.s_FormatoActualTabla
    Label (447,203 487x36), "MODELO"
    Label (1111,203 156x36), "FORMATO"
    Label (1386,203 156x36), "ESPESOR"
    Label (46,203 199x36), "PRODUCIDAS"
    Rectangle (49,232 248x40), "%s", text variable: FuncParoNodoLocalCorteH3.Funci_CortHum3.Cont_Piezas_Ftc
    Rectangle (1578,261 274x3)
    Ellipse (1578,214 274x54), "FINALIZAR MODELO"
        OnMouseClick: OpenDialog Dialog=V_Emerg_Fin_Prod_Ch3, OpenModal=True, OpenCentered=True
    Label (46,332 390x54), "TURNO ACTUAL"
    Label (58,386 199x36), "PRODUCCIÓN"
    Label (731,457 261x36), "PARO ACTUAL", invisible if: FuncParoNodoLocalCorteH3.Funci_CortHum3.M_SinParo_Ftc
    Label (1240,453 261x36), "HORA INICIO", invisible if: FuncParoNodoLocalCorteH3.Funci_CortHum3.M_SinParo_Ftc
    RoundedRectangle (735,593 264x80), "DESCANSO", invisible if: FuncParoNodoLocalCorteH3.Funci_CortHum3.M_SinParo_Ftc
        OnMouseClick: execute { FuncParoNodoLocalCorteH3.FunGeneCortHum3.IndexJustificacionParo:=1; FuncParoNodoLocalCorteH3.FunGeneCortHum3.ListadoJustificacionParo(); }
    RoundedRectangle (1019,593 264x80), "AVERÍA", invisible if: FuncParoNodoLocalCorteH3.Funci_CortHum3.M_SinParo_Ftc
        OnMouseClick: execute { FuncParoNodoLocalCorteH3.FunGeneCortHum3.IndexJustificacionParo:=2; FuncParoNodoLocalCorteH3.FunGeneCortHum3.ListadoJustificacionParo(); }
    RoundedRectangle (1303,593 264x80), "CAMBIO DISCOS", invisible if: FuncParoNodoLocalCorteH3.Funci_CortHum3.M_SinParo_Ftc
        OnMouseClick: execute { FuncParoNodoLocalCorteH3.FunGeneCortHum3.IndexJustificacionParo:=3; FuncParoNodoLocalCorteH3.FunGeneCortHum3.ListadoJustificacionParo(); }
    RoundedRectangle (1587,593 264x80), "CAMBIO FORMATO", invisible if: FuncParoNodoLocalCorteH3.Funci_CortHum3.M_SinParo_Ftc
        OnMouseClick: execute { FuncParoNodoLocalCorteH3.FunGeneCortHum3.IndexJustificacionParo:=4; FuncParoNodoLocalCorteH3.FunGeneCortHum3.ListadoJustificacionParo(); }
    Rectangle (79,444 183x88), "%s", text variable: FuncParoNodoLocalCorteH3.Funci_CortHum3.Cont_Piezas_Ftc
    Label (216,487 106x36), "PIEZAS"
    Rectangle (216,518 96x4), colour toggle: FuncParoNodoLocalCorteH3.Funci_CortHum3.Fotocelula
    Label (731,528 261x36), "JUSTIFICAR PARO", invisible if: FuncParoNodoLocalCorteH3.Funci_CortHum3.M_SinParo_Ftc
    Rectangle (714,424 1164x4), invisible if: FuncParoNodoLocalCorteH3.Funci_CortHum3.M_SinParo_Ftc
    Rectangle (710,380 371x48), invisible if: FuncParoNodoLocalCorteH3.Funci_CortHum3.M_SinParo_Ftc
    Label (731,391 199x36), "PAROS", invisible if: FuncParoNodoLocalCorteH3.Funci_CortHum3.M_SinParo_Ftc
    Label (865,393 326x30), "NINGÚN PARO ACTIVO", invisible if: FuncParoNodoLocalCorteH3.Funci_CortHum3.MParo_Ftc
    Label (865,393 235x30), "PARO ACTIVO", invisible if: FuncParoNodoLocalCorteH3.Funci_CortHum3.M_SinParo_Ftc
    Ellipse (538,25 163x48), "HISTÓRICO"
        OnMouseClick: change screen: HistTablaTablas_Ch2
    Label (130,555 367x36), "PARO TOTAL ACUMULADO"
    Rectangle (45,658 295x88), "%t[H'h'm'min']", text variable: FuncParoNodoLocalCorteH3.Funci_CortHum3.fbTiempParoAcumDiario.t_Acumulado
    Label (86,611 76x36), "Día"
    Image (-3,943 1927x139), image: Imagenes.NeolithHeader
    Rectangle (237,758 325x88), "%t[H'h'm'min']", text variable: FuncParoNodoLocalCorteH3.Funci_CortHum3.fbTiempParoAcumTurno.t_Acumulado
    Label (106,775 102x36), "Turno"
    Rectangle (362,661 388x88), "%t[H'h'm'min']", text variable: FuncParoNodoLocalCorteH3.Funci_CortHum3.fbTiempParoAcumModelo.t_Acumulado
    Label (469,609 118x36), "Modelo"
    RoundedRectangle (777,713 264x80), "MANTENIMIENTO", invisible if: FuncParoNodoLocalCorteH3.Funci_CortHum3.M_SinParo_Ftc
        OnMouseClick: execute { FuncParoNodoLocalCorteH3.FunGeneCortHum3.IndexJustificacionParo:=6; FuncParoNodoLocalCorteH3.FunGeneCortHum3.ListadoJustificacionParo(); }
    RoundedRectangle (1096,713 372x80), "FALTA DE MATERIAL", invisible if: FuncParoNodoLocalCorteH3.Funci_CortHum3.M_SinParo_Ftc
        OnMouseClick: execute { FuncParoNodoLocalCorteH3.FunGeneCortHum3.IndexJustificacionParo:=7; FuncParoNodoLocalCorteH3.FunGeneCortHum3.ListadoJustificacionParo(); }
    RoundedRectangle (1504,713 368x80), "PREPARACION MATERIAL", invisible if: FuncParoNodoLocalCorteH3.Funci_CortHum3.M_SinParo_Ftc
        OnMouseClick: execute { FuncParoNodoLocalCorteH3.FunGeneCortHum3.IndexJustificacionParo:=8; FuncParoNodoLocalCorteH3.FunGeneCortHum3.ListadoJustificacionParo(); }
    RoundedRectangle (1032,503 389x80), "LIMPIEZA FIN DE TURNO", invisible if: FuncParoNodoLocalCorteH3.Funci_CortHum3.M_SinParo_Ftc
        OnMouseClick: execute { FuncParoNodoLocalCorteH3.FunGeneCortHum3.IndexJustificacionParo:=9; FuncParoNodoLocalCorteH3.FunGeneCortHum3.ListadoJustificacionParo(); }
END_VISUALIZATION

// ---- VISUs/Home_Sel_Maq.TcVIS
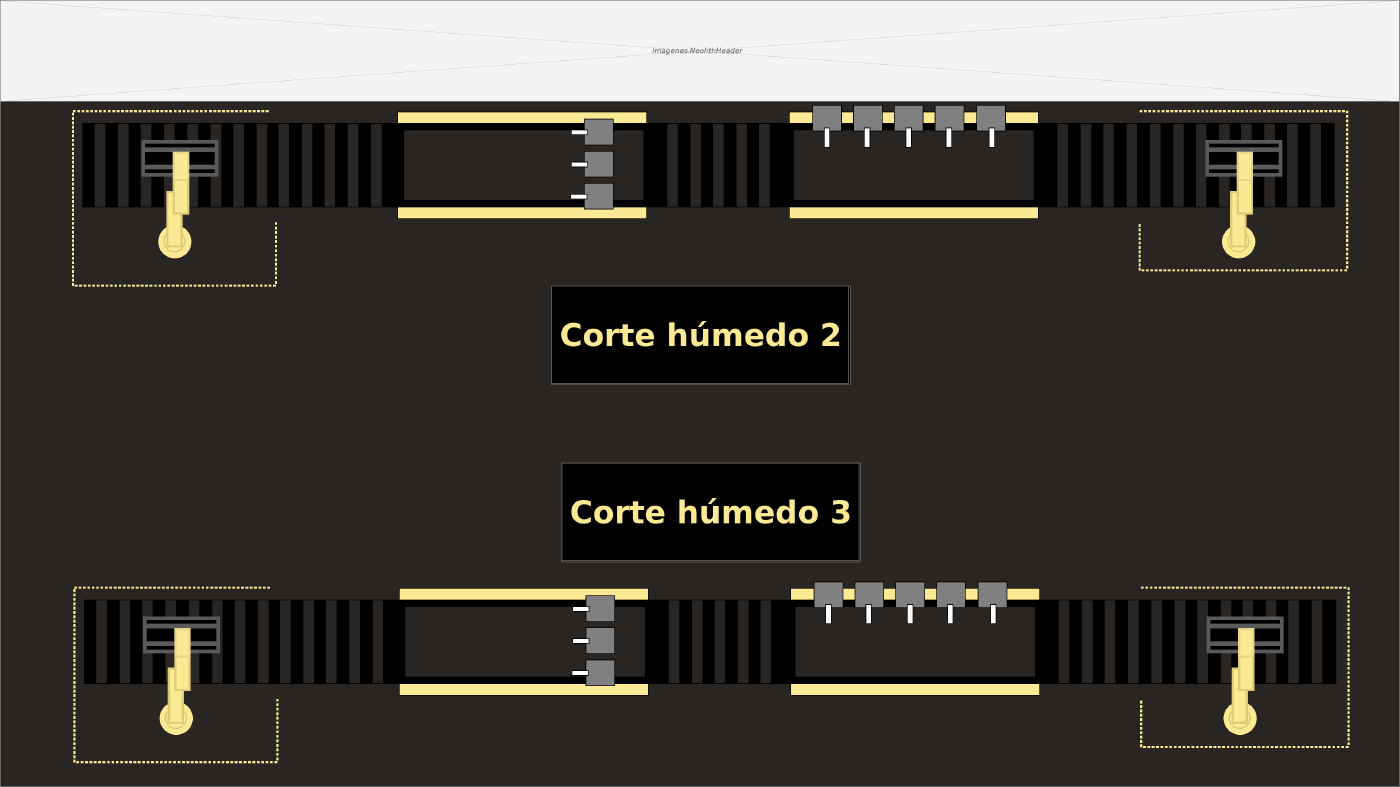
VISUALIZATION Home_Sel_Maq  // 1920x1080
    Button (756,392 410x136), "Corte húmedo 2"
        OnMouseUp: change screen: Home_CortH2
    Button (770,635 410x136), "Corte húmedo 3"
        OnMouseUp: change screen: Home_CortH3
    Image (-7,0 1927x139), image: Imagenes.NeolithHeader
    Group (100,144 1747x248)
        Rectangle (445,9 342x147)
        Rectangle (982,9 342x147)
        Rectangle (13,25 1717x115)
        Group (1349,25 363x115)
            Rectangle (0,0 16x115)
            Rectangle (32,0 16x115)
            Group (63,0 48x115)
                Rectangle (0,0 16x115)
                Rectangle (32,0 16x115)
            Group (127,0 111x115)
                Rectangle (0,0 16x115)
                Rectangle (32,0 16x115)
                Group (63,0 48x115)
                    Rectangle (0,0 16x115)
                    Rectangle (32,0 16x115)
            Rectangle (252,0 16x115)
            Rectangle (284,0 16x115)
            Group (315,0 48x115)
                Rectangle (0,0 16x115)
                Rectangle (32,0 16x115)
        Group (29,25 363x115)
            Rectangle (0,0 16x115)
            Rectangle (32,0 16x115)
            Group (63,0 48x115)
                Rectangle (0,0 16x115)
                Rectangle (32,0 16x115)
            Group (127,0 111x115)
                Rectangle (0,0 16x115)
                Rectangle (32,0 16x115)
                Group (63,0 48x115)
                    Rectangle (0,0 16x115)
                    Rectangle (32,0 16x115)
            Rectangle (252,0 16x115)
            Rectangle (284,0 16x115)
            Group (315,0 48x115)
                Rectangle (0,0 16x115)
                Rectangle (32,0 16x115)
        Rectangle (408,25 16x115)
        Rectangle (453,34 330x97)
        Rectangle (701,19 40x36)
        Rectangle (701,63 40x36)
        Rectangle (701,107 40x36)
        Rectangle (683,34 23x7)
        Rectangle (683,78 23x7)
        Rectangle (682,122 23x7)
        Rectangle (988,34 330x97)
        Rectangle (1014,0 40x36)
        Rectangle (1070,0 40x36)
        Rectangle (1126,0 40x36)
        Rectangle (1182,0 40x36)
        Rectangle (1239,0 40x36)
        Rectangle (1085,31 8x27)
        Rectangle (1030,31 8x27)
        Rectangle (1142,31 8x27)
        Rectangle (1197,31 8x27)
        Rectangle (1256,31 8x27)
        Group (814,25 142x115)
            Rectangle (126,0 16x115)
            Rectangle (0,0 16x115)
            Rectangle (32,0 16x115)
            Group (63,0 48x115)
                Rectangle (0,0 16x115)
                Rectangle (32,0 16x115)
        Polyline (1463,8) (1747,8) (1747,227) (1463,227) (1463,161)
        Polyline (278,161) (278,248) (0,248) (0,8) (271,8)
        Group (94,48 105x162)
            Ellipse (23,117 45x45)
            Ellipse (30,124 30x30)
            RoundedRectangle (34,70 22x77)
            RoundedRectangle (0,0 105x50)
            Rectangle (0,10 105x6)
            Rectangle (0,34 105x6)
            RoundedRectangle (43,25 22x77)
            RoundedRectangle (43,16 22x40)
        Group (1553,48 105x162)
            Ellipse (23,117 45x45)
            Ellipse (30,124 30x30)
            RoundedRectangle (34,70 22x77)
            RoundedRectangle (0,0 105x50)
            Rectangle (0,10 105x6)
            Rectangle (0,34 105x6)
            RoundedRectangle (43,25 22x77)
            RoundedRectangle (43,16 22x40)
    Group (102,798 1747x248)
        Rectangle (445,9 342x147)
        Rectangle (982,9 342x147)
        Rectangle (13,25 1717x115)
        Group (1349,25 363x115)
            Rectangle (0,0 16x115)
            Rectangle (32,0 16x115)
            Group (63,0 48x115)
                Rectangle (0,0 16x115)
                Rectangle (32,0 16x115)
            Group (127,0 111x115)
                Rectangle (0,0 16x115)
                Rectangle (32,0 16x115)
                Group (63,0 48x115)
                    Rectangle (0,0 16x115)
                    Rectangle (32,0 16x115)
            Rectangle (252,0 16x115)
            Rectangle (284,0 16x115)
            Group (315,0 48x115)
                Rectangle (0,0 16x115)
                Rectangle (32,0 16x115)
        Group (29,25 363x115)
            Rectangle (0,0 16x115)
            Rectangle (32,0 16x115)
            Group (63,0 48x115)
                Rectangle (0,0 16x115)
                Rectangle (32,0 16x115)
            Group (127,0 111x115)
                Rectangle (0,0 16x115)
                Rectangle (32,0 16x115)
                Group (63,0 48x115)
                    Rectangle (0,0 16x115)
                    Rectangle (32,0 16x115)
            Rectangle (252,0 16x115)
            Rectangle (284,0 16x115)
            Group (315,0 48x115)
                Rectangle (0,0 16x115)
                Rectangle (32,0 16x115)
        Rectangle (408,25 16x115)
        Rectangle (453,34 330x97)
        Rectangle (701,19 40x36)
        Rectangle (701,63 40x36)
        Rectangle (701,107 40x36)
        Rectangle (683,34 23x7)
        Rectangle (683,78 23x7)
        Rectangle (682,122 23x7)
        Rectangle (988,34 330x97)
        Rectangle (1014,0 40x36)
        Rectangle (1070,0 40x36)
        Rectangle (1126,0 40x36)
        Rectangle (1182,0 40x36)
        Rectangle (1239,0 40x36)
        Rectangle (1085,31 8x27)
        Rectangle (1030,31 8x27)
        Rectangle (1142,31 8x27)
        Rectangle (1197,31 8x27)
        Rectangle (1256,31 8x27)
        Group (814,25 142x115)
            Rectangle (126,0 16x115)
            Rectangle (0,0 16x115)
            Rectangle (32,0 16x115)
            Group (63,0 48x115)
                Rectangle (0,0 16x115)
                Rectangle (32,0 16x115)
        Polyline (1463,8) (1747,8) (1747,227) (1463,227) (1463,161)
        Polyline (278,161) (278,248) (0,248) (0,8) (271,8)
        Group (94,48 105x162)
            Ellipse (23,117 45x45)
            Ellipse (30,124 30x30)
            RoundedRectangle (34,70 22x77)
            RoundedRectangle (0,0 105x50)
            Rectangle (0,10 105x6)
            Rectangle (0,34 105x6)
            RoundedRectangle (43,25 22x77)
            RoundedRectangle (43,16 22x40)
        Group (1553,48 105x162)
            Ellipse (23,117 45x45)
            Ellipse (30,124 30x30)
            RoundedRectangle (34,70 22x77)
            RoundedRectangle (0,0 105x50)
            Rectangle (0,10 105x6)
            Rectangle (0,34 105x6)
            RoundedRectangle (43,25 22x77)
            RoundedRectangle (43,16 22x40)
END_VISUALIZATION

// ---- VISUs/Listas_Para_Desplegables/FormatoTabla.TcTLO
TEXTLIST FormatoTabla
  0 = 'Sin seleccionar'
  1 = '3200 X 1500'
  2 = '3600 X 1200'
  3 = '1800 X 1200'
  4 = '3000 X 1000'
  5 = '2600 X 1500'
  6 = '800 X 700'
  7 = '2700 X 1000'
  8 = 'Ninguno de la lista'
   = ''
END_TEXTLIST

// ---- VISUs/Listas_Para_Desplegables/EspesorTabla.TcTLO
TEXTLIST EspesorTabla
  0 = 'Sin seleccionar'
  1 = '3'
  2 = '6'
  3 = '12'
  4 = '20'
   = ''
END_TEXTLIST

// ---- VISUs/Modelo_Tabla_Ch2.TcVIS
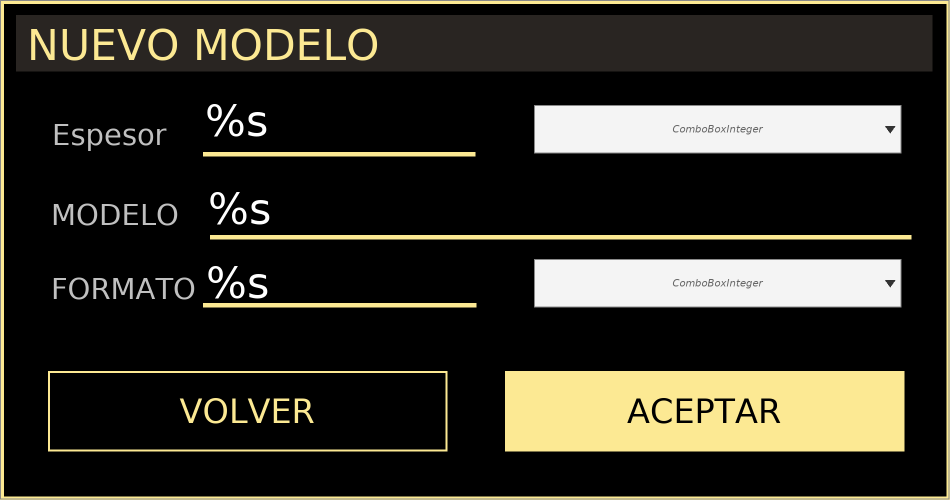
VISUALIZATION Modelo_Tabla_Ch2  // 950x500
    Rectangle (16,15 916x56)
    Rectangle (0,0 950x500)
    Label (24,17 498x56), "NUEVO MODELO"
    Rectangle (136,1125 690x58), "%s Contador piezas corte húmedo 4", text variable: FuncParoNodoRemote1CorteH2.Funci_CortHum2.Min_Parado_Ftc
    Button (871,1105 269x91), "Reset contador"
        tap FuncParoNodoRemote1CorteH2.Funci_CortHum2.ResetContPiez
    Rectangle (205,185 701x48), "%s", text variable: FuncParoNodoRemote1CorteH2.FunGeneCortHum2.s_ModeloEleccionTabla
        OnMouseDown: write the text variable via Edit
    Label (48,197 148x36), "MODELO"
    Rectangle (210,235 701x4)
    ComboBoxInteger (534,259 367x48), variable: FuncParoNodoRemote1CorteH2.FunGeneCortHum2.IndexListFormatoTabla, text list: 'FormatoTabla'
        p1601986498: ''
    Group (48,259 428x48), text variable: FuncParoNodoRemote1CorteH2.FunGeneCortHum2.s_FormatoEleccionTabla, input disabled if: FuncParoNodoRemote1CorteH2.FunGeneCortHum2.IndexListFormatoTabla<>6
        OnMouseClick: write the text variable via Edit
        Rectangle (155,0 273x48), "%s", text variable: FuncParoNodoRemote1CorteH2.sFormatoActualTabla
            OnMouseDown: write the text variable via Edit
        Label (0,12 148x36), "FORMATO"
        Rectangle (155,44 273x4)
    Rectangle (505,371 399x80), "ACEPTAR"
        tap FuncParoNodoRemote1CorteH2.FunGeneCortHum2.P_EscribirModelo
        OnMouseClick: CloseDialog Dialog=Modelo_Tabla_Ch2, Result=OK, NumpadKeypadSet=True
    Rectangle (48,371 399x80), "VOLVER"
        OnMouseClick: CloseDialog Dialog=Modelo_Tabla_Ch2, Result=None, NumpadKeypadSet=True
    Label (49,117 148x36), "Espesor"
    Rectangle (203,152 272x4)
    Rectangle (202,97 272x48), "%s", text variable: FuncParoNodoRemote1CorteH2.FunGeneCortHum2.s_EspesorEleccionTabla, input disabled if: FuncParoNodoRemote1CorteH2.FunGeneCortHum2.IndexListEsTabla<>6
        OnMouseDown: write the text variable via Edit
    ComboBoxInteger (534,105 367x48), variable: FuncParoNodoRemote1CorteH2.FunGeneCortHum2.IndexListEspesorTabla, input disabled if: FuncParoNodoRemote1CorteH2.FunGeneCortHum2.IndexListEsTabla<>6, text list: 'EspesorTabla'
        p1601986498: ''
END_VISUALIZATION

// ---- VISUs/Modelo_Tabla_Ch3.TcVIS
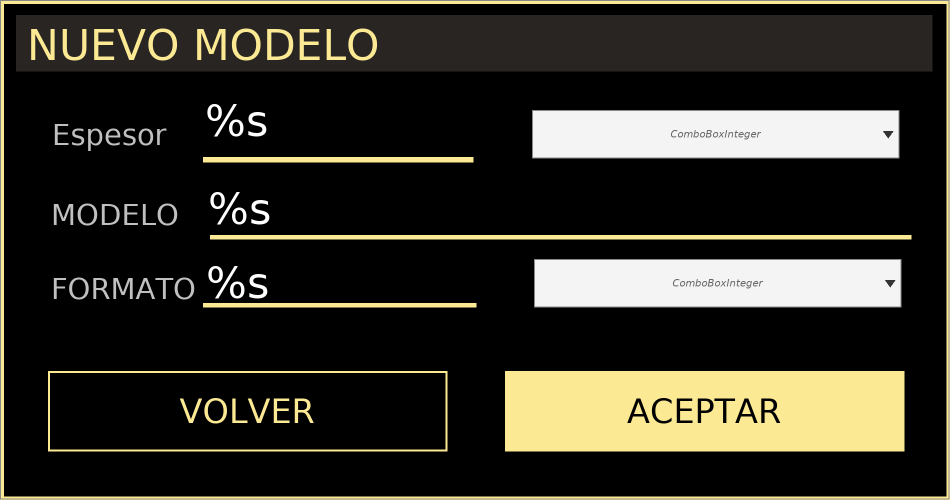
VISUALIZATION Modelo_Tabla_Ch3  // 950x500
    Rectangle (16,15 916x56)
    Rectangle (0,0 950x500)
    Label (24,17 498x56), "NUEVO MODELO"
    Rectangle (136,1125 690x58), "%s Contador piezas corte húmedo 4", text variable: FuncParoNodoRemote1CorteH2.CortHum2StrFuncParoEnviar.Cont_Piezas
    Button (871,1105 269x91), "Reset contador"
        tap FuncParoNodoLocalCorteH3.Funci_CortHum3.ResetContPiez
    ComboBoxInteger (534,259 367x48), variable: FuncParoNodoLocalCorteH3.FunGeneCortHum3.IndexListFormatoTabla, text list: 'FormatoTabla'
        p1601986498: ''
    Rectangle (205,185 701x48), "%s", text variable: FuncParoNodoLocalCorteH3.FunGeneCortHum3.s_ModeloEleccionTabla
        OnMouseDown: write the text variable via Edit
    Label (48,197 148x36), "MODELO"
    Rectangle (210,235 701x4)
    Rectangle (203,259 273x48), "%s", text variable: FuncParoNodoLocalCorteH3.sFormatoActualTabla, input disabled if: FuncParoNodoLocalCorteH3.FunGeneCortHum3.IndexListFormatoTabla<>6
        OnMouseDown: write the text variable via Edit
    Label (48,271 148x36), "FORMATO"
    Rectangle (203,303 273x4)
    Rectangle (505,371 399x80), "ACEPTAR"
        tap FuncParoNodoLocalCorteH3.FunGeneCortHum3.P_EscribirModelo
        OnMouseClick: CloseDialog Dialog=Modelo_Tabla_Ch3, Result=None, NumpadKeypadSet=True
    Rectangle (48,371 399x80), "VOLVER"
        OnMouseClick: CloseDialog Dialog=V_Emerg_Fin_Prod_Ch3, Result=None, NumpadKeypadSet=True
    Label (49,117 148x36), "Espesor"
    Rectangle (203,157 270x5)
    Rectangle (202,97 270x48), "%s", text variable: FuncParoNodoLocalCorteH3.FunGeneCortHum3.s_EspesorEleccionTabla, input disabled if: FuncParoNodoLocalCorteH3.FunGeneCortHum3.IndexListEspesorTabla<>6
        OnMouseDown: write the text variable via Edit
    ComboBoxInteger (532,110 367x48), variable: FuncParoNodoLocalCorteH3.FunGeneCortHum3.IndexListEspesorTabla, input disabled if: FuncParoNodoLocalCorteH3.FunGeneCortHum3.IndexListEspesorTabla<>6, text list: 'EspesorTabla'
        p1601986498: ''
END_VISUALIZATION

// ---- VISUs/V_Emerg_Fin_Prod_Ch2.TcVIS
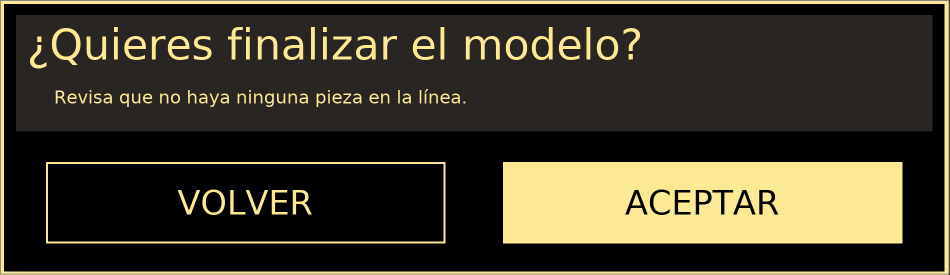
VISUALIZATION V_Emerg_Fin_Prod_Ch2  // 950x275
    Rectangle (0,0 948x275)
    Rectangle (16,15 916x116)
    Label (24,17 898x65), "¿Quieres finalizar el modelo?"
    Label (51,85 857x43), "Revisa que no haya ninguna pieza en la línea."
    Rectangle (503,162 399x81), "ACEPTAR"
        tap FuncParoNodoRemote1CorteH2.FunGeneCortHum2.P_FinProduccion
        OnMouseClick: CloseDialog Dialog=V_Emerg_Fin_Prod_Ch2, Result=None, NumpadKeypadSet=True
        OnMouseClick: OpenDialog Dialog=Modelo_Tabla_Ch2, OpenModal=True, OpenCentered=True
    Rectangle (46,162 399x81), "VOLVER"
        OnMouseClick: CloseDialog Dialog=V_Emerg_Fin_Prod_Ch2, Result=Cancel, NumpadKeypadSet=True
END_VISUALIZATION

// ---- VISUs/V_Emerg_Fin_Prod_Ch3.TcVIS
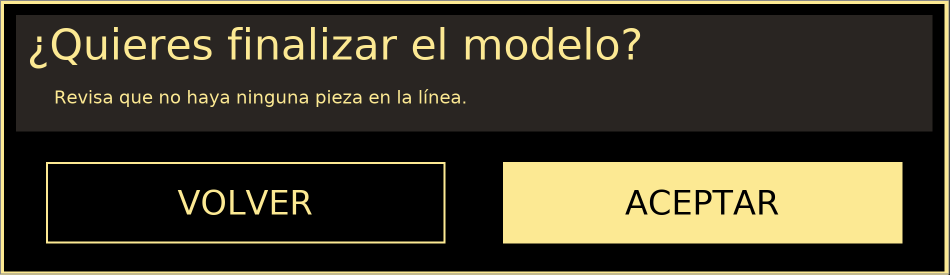
VISUALIZATION V_Emerg_Fin_Prod_Ch3  // 950x275
    Rectangle (0,0 948x275)
    Rectangle (16,15 916x116)
    Label (24,17 898x65), "¿Quieres finalizar el modelo?"
    Label (51,85 857x43), "Revisa que no haya ninguna pieza en la línea."
    Rectangle (503,162 399x81), "ACEPTAR"
        tap FuncParoNodoLocalCorteH3.FunGeneCortHum3.P_FinProduccion
        OnMouseClick: CloseDialog Dialog=V_Emerg_Fin_Prod_Ch3, Result=None, NumpadKeypadSet=True
        OnMouseClick: OpenDialog Dialog=Modelo_Tabla_Ch3, OpenModal=True, OpenCentered=True
    Rectangle (46,162 399x81), "VOLVER"
        OnMouseClick: CloseDialog Dialog=V_Emerg_Fin_Prod_Ch3, Result=None, NumpadKeypadSet=True
END_VISUALIZATION
